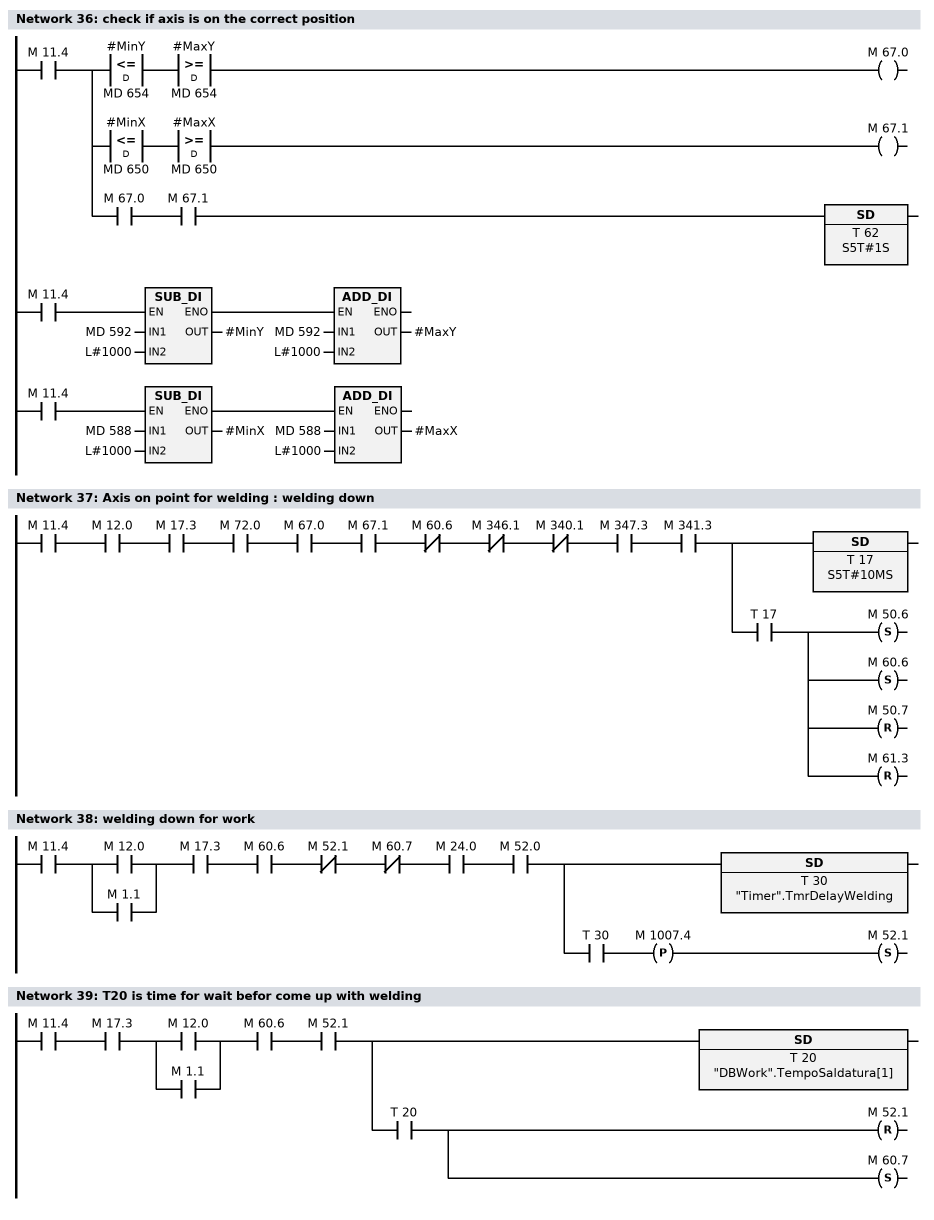
[picture p191: FC14 - AUTOMATIC networks 36-39]
NETWORK
TITLE = check if axis is on the correct position
      A     M 11.4;
      =     L 16.0;
      A(;
      A     L 16.0;
      JNB   _00e;
      L     MD 592;
      L     L#1000;
      -D;
      T     #MinY;
      AN    OV;
      SAVE;
      CLR;
_00e: A     BR;
      );
      JNB   _00f;
      L     MD 592;
      L     L#1000;
      +D;
      T     #MaxY;
_00f: NOP   0;
      A(;
      A     L 16.0;
      JNB   _010;
      L     MD 588;
      L     L#1000;
      -D;
      T     #MinX;
      AN    OV;
      SAVE;
      CLR;
_010: A     BR;
      );
      JNB   _011;
      L     MD 588;
      L     L#1000;
      +D;
      T     #MaxX;
_011: NOP   0;
      A     L 16.0;
      A(;
      L     #MinY;
      L     MD 654;
      <=D;
      );
      A(;
      L     #MaxY;
      L     MD 654;
      >=D;
      );
      =     M 67.0;
      A     L 16.0;
      A(;
      L     #MinX;
      L     MD 650;
      <=D;
      );
      A(;
      L     #MaxX;
      L     MD 650;
      >=D;
      );
      =     M 67.1;
      A     L 16.0;
      A     M 67.0;
      A     M 67.1;
      L     S5T#1S;
      SD    T 62;
NETWORK
TITLE = Axis on point for welding : welding down
//Saldatore giù
      A     M 11.4;
      A     M 12.0;
      A     M 17.3;
      A     M 72.0;
      A     M 67.0;
      A     M 67.1;
      AN    M 60.6;
      AN    M 346.1;
      AN    M 340.1;
      A     M 347.3;
      A     M 341.3;
      =     L 16.0;
      A     L 16.0;
      BLD   102;
      L     S5T#10MS;
      SD    T 17;
      A     L 16.0;
      A     T 17;
      S     M 50.6;
      S     M 60.6;
      R     M 50.7;
      R     M 61.3;
NETWORK
TITLE = welding down for work
//saldatore giu per saldatura
      A     M 11.4;
      A(;
      O     M 12.0;
      O     M 1.1;
      );
      A     M 17.3;
      A     M 60.6;
      AN    M 52.1;
      AN    M 60.7;
      A     M 24.0;
      A     M 52.0;
      =     L 16.0;
      A     L 16.0;
      BLD   102;
      L     "Timer".TmrDelayWelding;
      SD    T 30;
      A     L 16.0;
      A     T 30;
      FP    M 1007.4;
      S     M 52.1;
NETWORK
TITLE = T20 is time for wait befor come up with welding
//Resto un tempo T20 sul punto saldato prima di rialzare la torcia
      A     M 11.4;
      A     M 17.3;
      A(;
      O     M 12.0;
      O     M 1.1;
      );
      A     M 60.6;
      A     M 52.1;
      =     L 16.0;
      A     L 16.0;
      BLD   102;
      L     "DBWork".TempoSaldatura[1];
      SD    T 20;
      A     L 16.0;
      A     T 20;
      R     M 52.1;
      S     M 60.7;
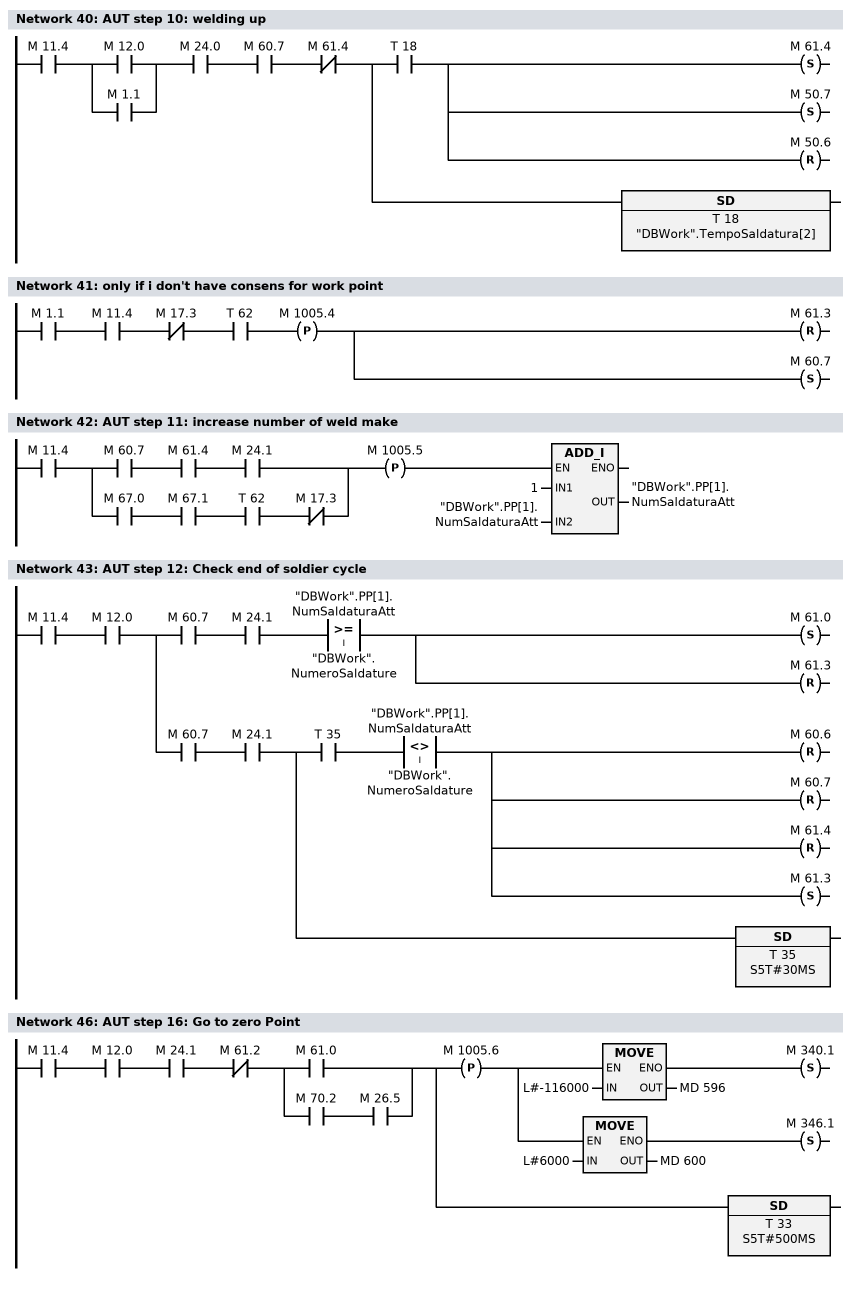
NETWORK
TITLE = AUT step 10: welding up
      A     M 11.4;
      A(;
      O     M 12.0;
      O     M 1.1;
      );
      A     M 24.0;
      A     M 60.7;
      AN    M 61.4;
      =     L 16.0;
      A     L 16.0;
      A     T 18;
      S     M 61.4;
      S     M 50.7;
      R     M 50.6;
      A     L 16.0;
      BLD   102;
      L     "DBWork".TempoSaldatura[2];
      SD    T 18;
NETWORK
TITLE = only if i don't have consens for work point
      A     M 1.1;
      A     M 11.4;
      AN    M 17.3;
      A     T 62;
      FP    M 1005.4;
      R     M 61.3;
      S     M 60.7;
NETWORK
TITLE = AUT step 11: increase number of weld make
//incremento il numero di saldature effettuate
      A     M 11.4;
      A(;
      A     M 60.7;
      A     M 61.4;
      A     M 24.1;
      O;
      A     M 67.0;
      A     M 67.1;
      A     T 62;
      AN    M 17.3;
      );
      FP    M 1005.5;
      JNB   _012;
      L     1;
      L     "DBWork".PP[1].NumSaldaturaAtt;
      +I;
      T     "DBWork".PP[1].NumSaldaturaAtt;
_012: NOP   0;
NETWORK
TITLE = AUT step 12: Check end of soldier cycle 
//aspetto per il passaggio delle coorddinate al simodrive
      A     M 11.4;
      A     M 12.0;
      =     L 16.0;
      A     L 16.0;
      A     M 60.7;
      A     M 24.1;
      A(;
      L     "DBWork".PP[1].NumSaldaturaAtt;
      L     "DBWork".NumeroSaldature;
      >=I;
      );
      S     M 61.0;
      R     M 61.3;
      A     L 16.0;
      A     M 60.7;
      A     M 24.1;
      =     L 16.1;
      A     L 16.1;
      A     T 35;
      A(;
      L     "DBWork".PP[1].NumSaldaturaAtt;
      L     "DBWork".NumeroSaldature;
      <>I;
      );
      R     M 60.6;
      R     M 60.7;
      R     M 61.4;
      S     M 61.3;
      A     L 16.1;
      BLD   102;
      L     S5T#30MS;
      SD    T 35;
NETWORK
TITLE =
NETWORK
TITLE =
NETWORK
TITLE = AUT step 16: Go to zero Point
      A     M 11.4;
      A     M 12.0;
      A     M 24.1;
      AN    M 61.2;
      A(;
      O     M 61.0;
      O;
      A     M 70.2;
      A     M 26.5;
      );
      =     L 16.0;
      A     L 16.0;
      FP    M 1005.6;
      =     L 16.1;
      A     L 16.1;
      JNB   _013;
      L     L#-116000;
      T     MD 596;
      SET;
      SAVE;
      CLR;
_013: A     BR;
      S     M 340.1;
      A     L 16.1;
      JNB   _014;
      L     L#6000;
      T     MD 600;
      SET;
      SAVE;
      CLR;
_014: A     BR;
      S     M 346.1;
      A     L 16.0;
      BLD   102;
      L     S5T#500MS;
      SD    T 33;
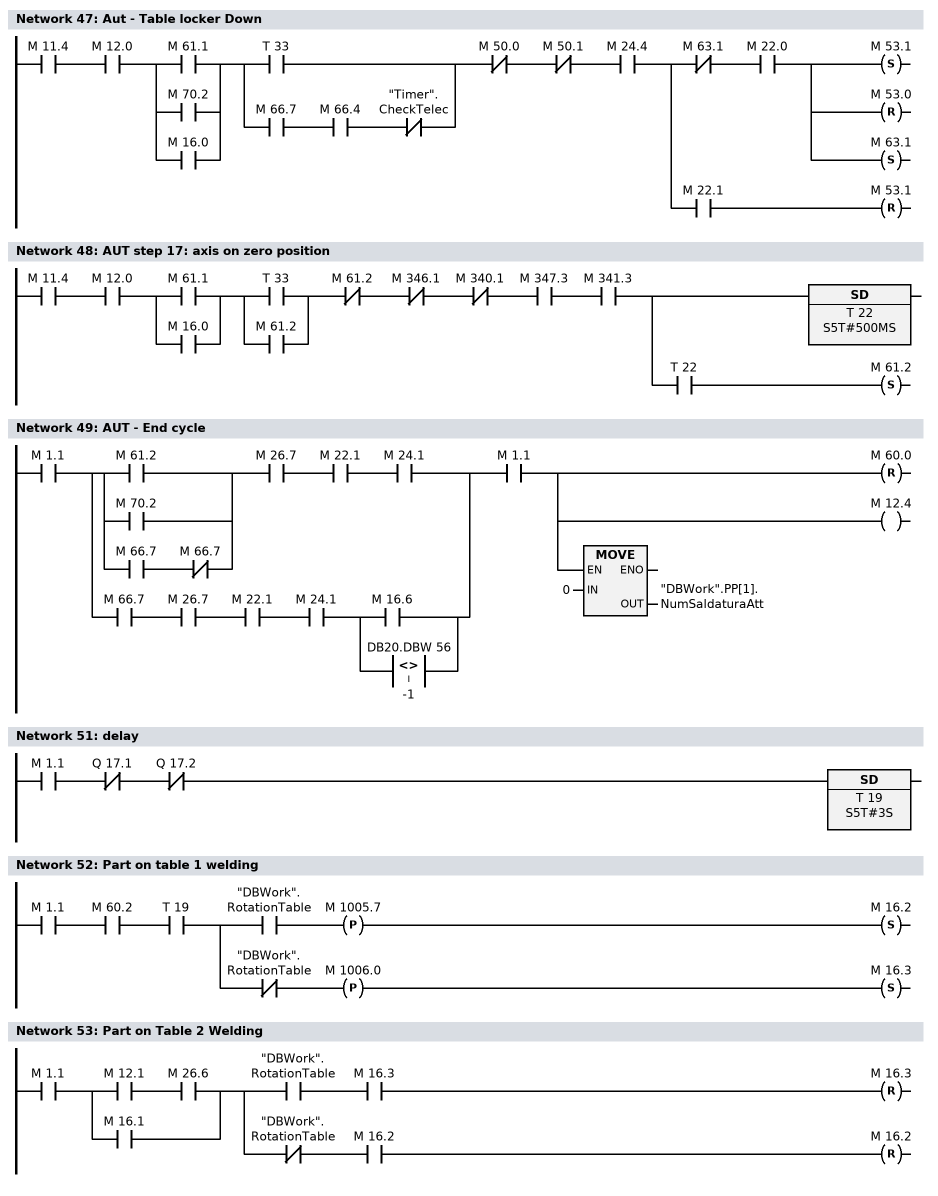
NETWORK
TITLE = Aut - Table locker Down
//Table cyclinder Low
      A     M 11.4;
      A     M 12.0;
      A(;
      O     M 61.1;
      O     M 70.2;
      O     M 16.0;
      );
      A(;
      O     T 33;
      O;
      A     M 66.7;
      A     M 66.4;
      AN    "Timer".CheckTelec;
      );
      AN    M 50.0;
      AN    M 50.1;
      A     M 24.4;
      =     L 16.0;
      A     L 16.0;
      AN    M 63.1;
      A     M 22.0;
      S     M 53.1;
      R     M 53.0;
      S     M 63.1;
      A     L 16.0;
      A     M 22.1;
      R     M 53.1;
NETWORK
TITLE = AUT step 17: axis on zero position
      A     M 11.4;
      A     M 12.0;
      A(;
      O     M 61.1;
      O     M 16.0;
      );
      A(;
      O     T 33;
      O     M 61.2;
      );
      AN    M 61.2;
      AN    M 346.1;
      AN    M 340.1;
      A     M 347.3;
      A     M 341.3;
      =     L 16.0;
      A     L 16.0;
      BLD   102;
      L     S5T#500MS;
      SD    T 22;
      A     L 16.0;
      A     T 22;
      S     M 61.2;
NETWORK
TITLE = AUT - End cycle
      A     M 1.1;
      A(;
      A(;
      O     M 61.2;
      O     M 70.2;
      O;
      A     M 66.7;
      AN    M 66.7;
      );
      A     M 26.7;
      A     M 22.1;
      A     M 24.1;
      O;
      A     M 66.7;
      A     M 26.7;
      A     M 22.1;
      A     M 24.1;
      A(;
      O     M 16.6;
      O(;
      L     DB20.DBW 56;
      L     -1;
      <>I;
      );
      );
      );
      A     M 1.1;
      =     L 16.0;
      A     L 16.0;
      BLD   102;
      R     M 60.0;
      A     L 16.0;
      BLD   102;
      =     M 12.4;
      A     L 16.0;
      JNB   _015;
      L     0;
      T     "DBWork".PP[1].NumSaldaturaAtt;
_015: NOP   0;
NETWORK
TITLE =
NETWORK
TITLE = delay
      A     M 1.1;
      AN    Q 17.1;
      AN    Q 17.2;
      L     S5T#3S;
      SD    T 19;
NETWORK
TITLE = Part on table 1 welding
      A     M 1.1;
      A     M 60.2;
      A     T 19;
      =     L 16.0;
      A     L 16.0;
      A     "DBWork".RotationTable;
      FP    M 1005.7;
      S     M 16.2;
      A     L 16.0;
      AN    "DBWork".RotationTable;
      FP    M 1006.0;
      S     M 16.3;
NETWORK
TITLE = Part on Table 2 Welding
      A     M 1.1;
      A(;
      A     M 12.1;
      A     M 26.6;
      O     M 16.1;
      );
      =     L 16.0;
      A     L 16.0;
      A     "DBWork".RotationTable;
      A     M 16.3;
      R     M 16.3;
      A     L 16.0;
      AN    "DBWork".RotationTable;
      A     M 16.2;
      R     M 16.2;
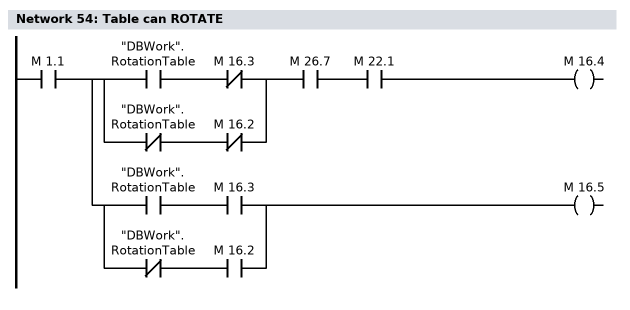
NETWORK
TITLE = Table can ROTATE
      A     M 1.1;
      =     L 16.0;
      A     L 16.0;
      A(;
      A     "DBWork".RotationTable;
      AN    M 16.3;
      O;
      AN    "DBWork".RotationTable;
      AN    M 16.2;
      );
      A     M 26.7;
      A     M 22.1;
      =     M 16.4;
      A     L 16.0;
      A(;
      A     "DBWork".RotationTable;
      A     M 16.3;
      O;
      AN    "DBWork".RotationTable;
      A     M 16.2;
      );
      =     M 16.5;
END_FUNCTION

FUNCTION "FC16 - ALARMS" : VOID	// FC 16
TITLE = Alarms management
VERSION : 0.1
VAR_TEMP
  tempBOOL : BOOL ;
END_VAR
BEGIN
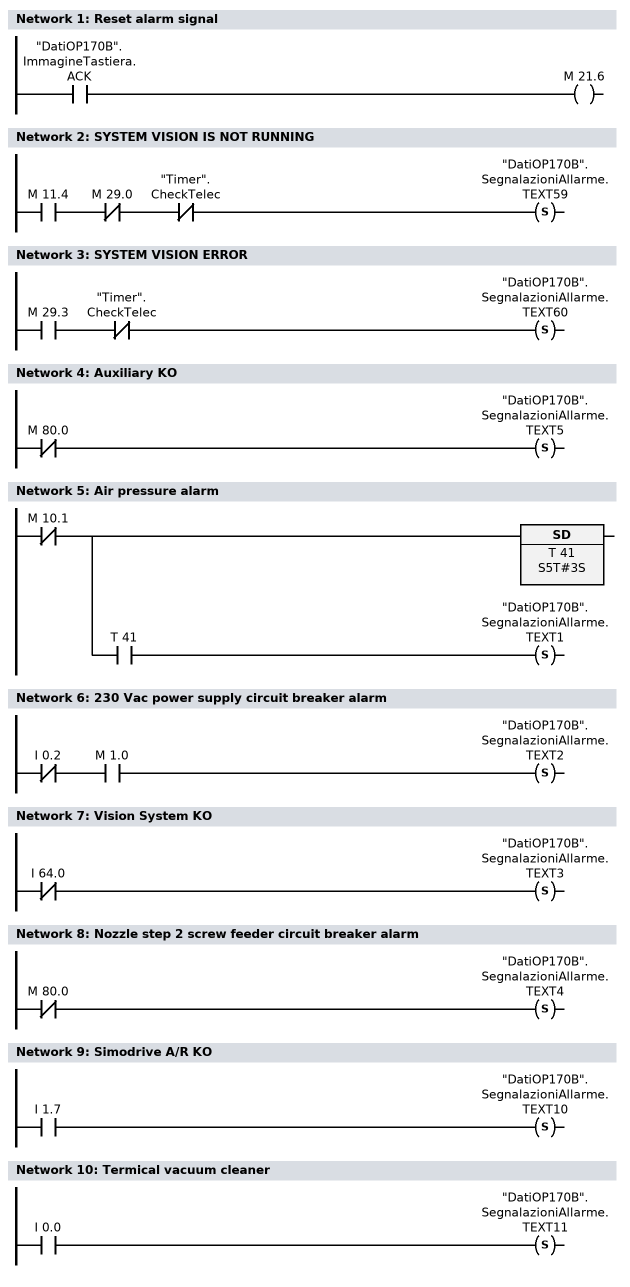
NETWORK
TITLE = Reset alarm signal
      A     "DatiOP170B".ImmagineTastiera.ACK;
      =     M 21.6;
NETWORK
TITLE = SYSTEM VISION IS NOT RUNNING
      A     M 11.4;
      AN    M 29.0;
      AN    "Timer".CheckTelec;
      S     "DatiOP170B".SegnalazioniAllarme.TEXT59;
NETWORK
TITLE = SYSTEM VISION ERROR
      A     M 29.3;
      AN    "Timer".CheckTelec;
      S     "DatiOP170B".SegnalazioniAllarme.TEXT60;
NETWORK
TITLE = Auxiliary KO
      AN    M 80.0;
      S     "DatiOP170B".SegnalazioniAllarme.TEXT5;
NETWORK
TITLE = Air pressure alarm
      AN    M 10.1;
      =     L 1.0;
      A     L 1.0;
      BLD   102;
      L     S5T#3S;
      SD    T 41;
      A     L 1.0;
      A     T 41;
      S     "DatiOP170B".SegnalazioniAllarme.TEXT1;
NETWORK
TITLE = 230 Vac power supply circuit breaker alarm
      AN    I 0.2;
      A     M 1.0;
      S     "DatiOP170B".SegnalazioniAllarme.TEXT2;
NETWORK
TITLE = Vision System KO
      AN    I 64.0;
      S     "DatiOP170B".SegnalazioniAllarme.TEXT3;
NETWORK
TITLE = Nozzle step 2 screw feeder circuit breaker alarm
      AN    M 80.0;
      S     "DatiOP170B".SegnalazioniAllarme.TEXT4;
NETWORK
TITLE = Simodrive A/R KO
      A     I 1.7;
      S     "DatiOP170B".SegnalazioniAllarme.TEXT10;
NETWORK
TITLE = Termical vacuum cleaner
      A     I 0.0;
      S     "DatiOP170B".SegnalazioniAllarme.TEXT11;
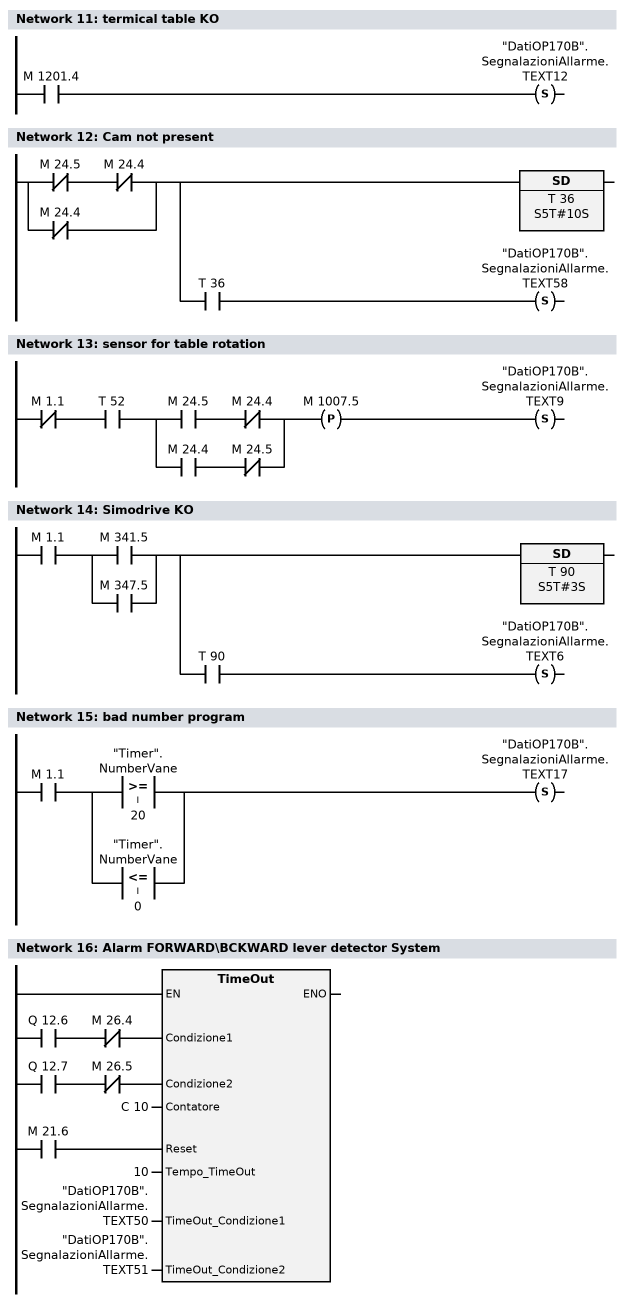
NETWORK
TITLE = termical table KO
      A     M 1201.4;
      S     "DatiOP170B".SegnalazioniAllarme.TEXT12;
NETWORK
TITLE = Cam not present
      AN    M 24.5;
      AN    M 24.4;
      ON    M 24.4;
      =     L 1.0;
      A     L 1.0;
      BLD   102;
      L     S5T#10S;
      SD    T 36;
      A     L 1.0;
      A     T 36;
      S     "DatiOP170B".SegnalazioniAllarme.TEXT58;
NETWORK
TITLE = sensor for table rotation
      AN    M 1.1;
      A     T 52;
      A(;
      A     M 24.5;
      AN    M 24.4;
      O;
      A     M 24.4;
      AN    M 24.5;
      );
      FP    M 1007.5;
      S     "DatiOP170B".SegnalazioniAllarme.TEXT9;
NETWORK
TITLE = Simodrive KO
//press ack button
      A     M 1.1;
      A(;
      O     M 341.5;
      O     M 347.5;
      );
      =     L 1.0;
      A     L 1.0;
      BLD   102;
      L     S5T#3S;
      SD    T 90;
      A     L 1.0;
      A     T 90;
      S     "DatiOP170B".SegnalazioniAllarme.TEXT6;
NETWORK
TITLE = bad number program
      A     M 1.1;
      A(;
      O(;
      L     "Timer".NumberVane;
      L     20;
      >=I;
      );
      O(;
      L     "Timer".NumberVane;
      L     0;
      <=I;
      );
      );
      S     "DatiOP170B".SegnalazioniAllarme.TEXT17;
NETWORK
TITLE = Alarm FORWARD\BCKWARD lever detector System
      A     Q 12.6;
      AN    M 26.4;
      =     L 1.0;
      BLD   103;
      A     Q 12.7;
      AN    M 26.5;
      =     L 1.1;
      BLD   103;
      A     M 21.6;
      =     L 1.2;
      BLD   103;
      CALL  "TimeOut" (
           Condizione1              := L 1.0,
           Condizione2              := L 1.1,
           Contatore                := C 10,
           Reset                    := L 1.2,
           Tempo_TimeOut            := 10,
           TimeOut_Condizione1      := "DatiOP170B".SegnalazioniAllarme.TEXT50,
           TimeOut_Condizione2      := "DatiOP170B".SegnalazioniAllarme.TEXT51);
      NOP   0;
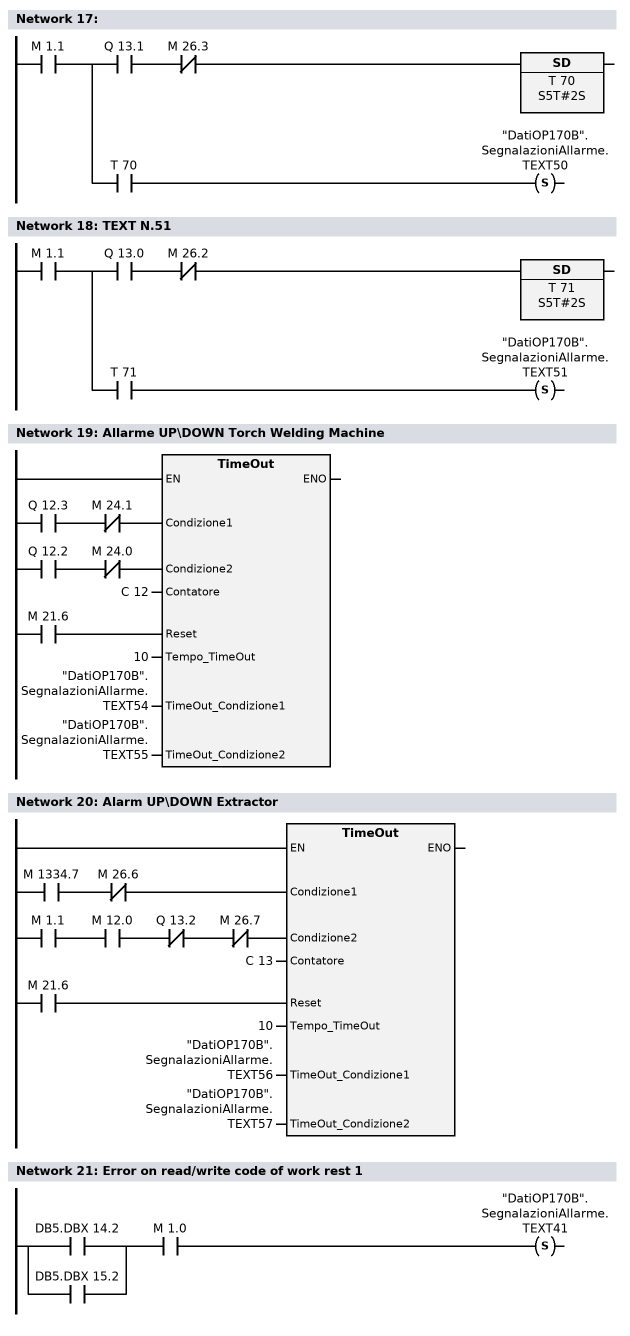
NETWORK
TITLE =
      A     M 1.1;
      =     L 1.0;
      A     L 1.0;
      A     Q 13.1;
      AN    M 26.3;
      L     S5T#2S;
      SD    T 70;
      A     L 1.0;
      A     T 70;
      S     "DatiOP170B".SegnalazioniAllarme.TEXT50;
NETWORK
TITLE = TEXT N.51
      A     M 1.1;
      =     L 1.0;
      A     L 1.0;
      A     Q 13.0;
      AN    M 26.2;
      L     S5T#2S;
      SD    T 71;
      A     L 1.0;
      A     T 71;
      S     "DatiOP170B".SegnalazioniAllarme.TEXT51;
NETWORK
TITLE = Allarme UP\DOWN Torch Welding Machine
      A     Q 12.3;
      AN    M 24.1;
      =     L 1.0;
      BLD   103;
      A     Q 12.2;
      AN    M 24.0;
      =     L 1.1;
      BLD   103;
      A     M 21.6;
      =     L 1.2;
      BLD   103;
      CALL  "TimeOut" (
           Condizione1              := L 1.0,
           Condizione2              := L 1.1,
           Contatore                := C 12,
           Reset                    := L 1.2,
           Tempo_TimeOut            := 10,
           TimeOut_Condizione1      := "DatiOP170B".SegnalazioniAllarme.TEXT54,
           TimeOut_Condizione2      := "DatiOP170B".SegnalazioniAllarme.TEXT55);
      NOP   0;
NETWORK
TITLE = Alarm UP\DOWN Extractor
      A     M 1334.7;
      AN    M 26.6;
      =     L 1.0;
      BLD   103;
      A     M 1.1;
      A     M 12.0;
      AN    Q 13.2;
      AN    M 26.7;
      =     L 1.1;
      BLD   103;
      A     M 21.6;
      =     L 1.2;
      BLD   103;
      CALL  "TimeOut" (
           Condizione1              := L 1.0,
           Condizione2              := L 1.1,
           Contatore                := C 13,
           Reset                    := L 1.2,
           Tempo_TimeOut            := 10,
           TimeOut_Condizione1      := "DatiOP170B".SegnalazioniAllarme.TEXT56,
           TimeOut_Condizione2      := "DatiOP170B".SegnalazioniAllarme.TEXT57);
      NOP   0;
NETWORK
TITLE = Error on read/write code of work rest 1
      A(;
      O     DB5.DBX 14.2;
      O     DB5.DBX 15.2;
      );
      A     M 1.0;
      S     "DatiOP170B".SegnalazioniAllarme.TEXT41;
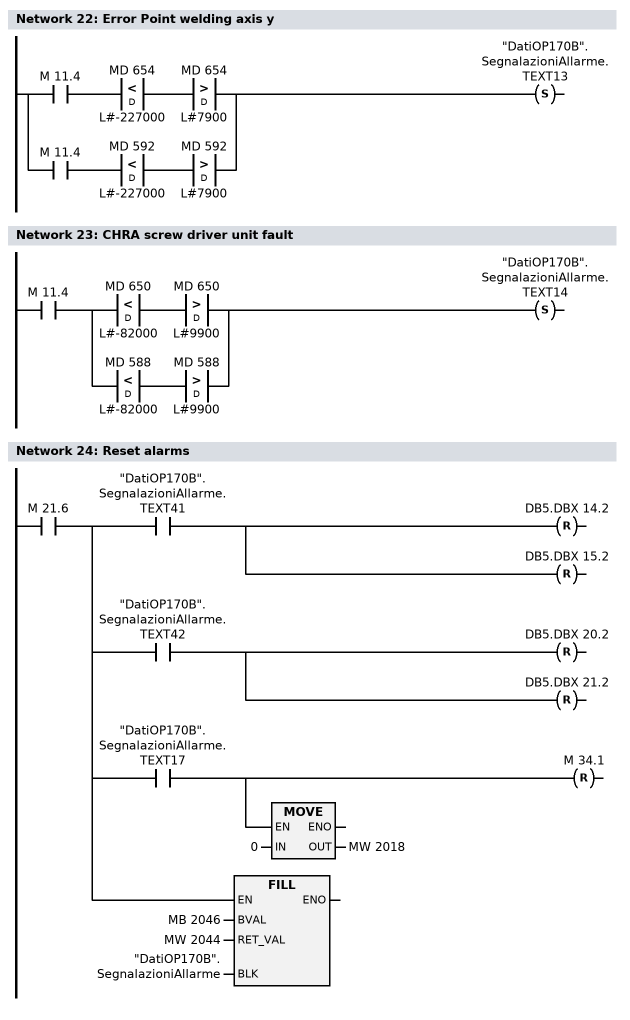
NETWORK
TITLE = Error Point welding axis y
      A     M 11.4;
      A(;
      L     MD 654;
      L     L#-227000;
      <D;
      );
      A(;
      L     MD 654;
      L     L#7900;
      >D;
      );
      O;
      A     M 11.4;
      A(;
      L     MD 592;
      L     L#-227000;
      <D;
      );
      A(;
      L     MD 592;
      L     L#7900;
      >D;
      );
      S     "DatiOP170B".SegnalazioniAllarme.TEXT13;
NETWORK
TITLE = CHRA screw driver unit fault
      A     M 11.4;
      A(;
      A(;
      L     MD 650;
      L     L#-82000;
      <D;
      );
      A(;
      L     MD 650;
      L     L#9900;
      >D;
      );
      O;
      A(;
      L     MD 588;
      L     L#-82000;
      <D;
      );
      A(;
      L     MD 588;
      L     L#9900;
      >D;
      );
      );
      S     "DatiOP170B".SegnalazioniAllarme.TEXT14;
NETWORK
TITLE = Reset alarms
      A     M 21.6;
      =     L 1.0;
      A     L 1.0;
      A     "DatiOP170B".SegnalazioniAllarme.TEXT41;
      R     DB5.DBX 14.2;
      R     DB5.DBX 15.2;
      A     L 1.0;
      A     "DatiOP170B".SegnalazioniAllarme.TEXT42;
      R     DB5.DBX 20.2;
      R     DB5.DBX 21.2;
      A     L 1.0;
      A     "DatiOP170B".SegnalazioniAllarme.TEXT17;
      =     L 1.1;
      A     L 1.1;
      BLD   102;
      R     M 34.1;
      A     L 1.1;
      JNB   _001;
      L     0;
      T     MW 2018;
_001: NOP   0;
      A     L 1.0;
      JNB   _002;
      CALL  "FILL" (
           BVAL                     := MB 2046,
           RET_VAL                  := MW 2044,
           BLK                      := "DatiOP170B".SegnalazioniAllarme);
_002: NOP   0;
NETWORK
TITLE = Spacer circular feeder empty
      CLR;
      =     "DatiOP170B".SegnalazioniAllarme.TEXT15;
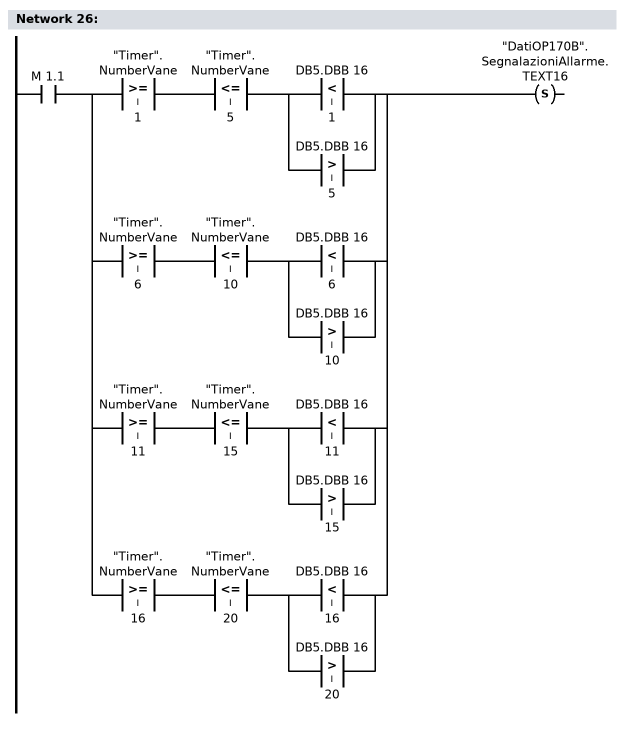
NETWORK
TITLE =
      A     M 1.1;
      A(;
      A(;
      L     "Timer".NumberVane;
      L     1;
      >=I;
      );
      A(;
      L     "Timer".NumberVane;
      L     5;
      <=I;
      );
      A(;
      O(;
      L     DB5.DBB 16;
      L     1;
      <I;
      );
      O(;
      L     DB5.DBB 16;
      L     5;
      >I;
      );
      );
      O;
      A(;
      L     "Timer".NumberVane;
      L     6;
      >=I;
      );
      A(;
      L     "Timer".NumberVane;
      L     10;
      <=I;
      );
      A(;
      O(;
      L     DB5.DBB 16;
      L     6;
      <I;
      );
      O(;
      L     DB5.DBB 16;
      L     10;
      >I;
      );
      );
      O;
      A(;
      L     "Timer".NumberVane;
      L     11;
      >=I;
      );
      A(;
      L     "Timer".NumberVane;
      L     15;
      <=I;
      );
      A(;
      O(;
      L     DB5.DBB 16;
      L     11;
      <I;
      );
      O(;
      L     DB5.DBB 16;
      L     15;
      >I;
      );
      );
      O;
      A(;
      L     "Timer".NumberVane;
      L     16;
      >=I;
      );
      A(;
      L     "Timer".NumberVane;
      L     20;
      <=I;
      );
      A(;
      O(;
      L     DB5.DBB 16;
      L     16;
      <I;
      );
      O(;
      L     DB5.DBB 16;
      L     20;
      >I;
      );
      );
      );
      S     "DatiOP170B".SegnalazioniAllarme.TEXT16;
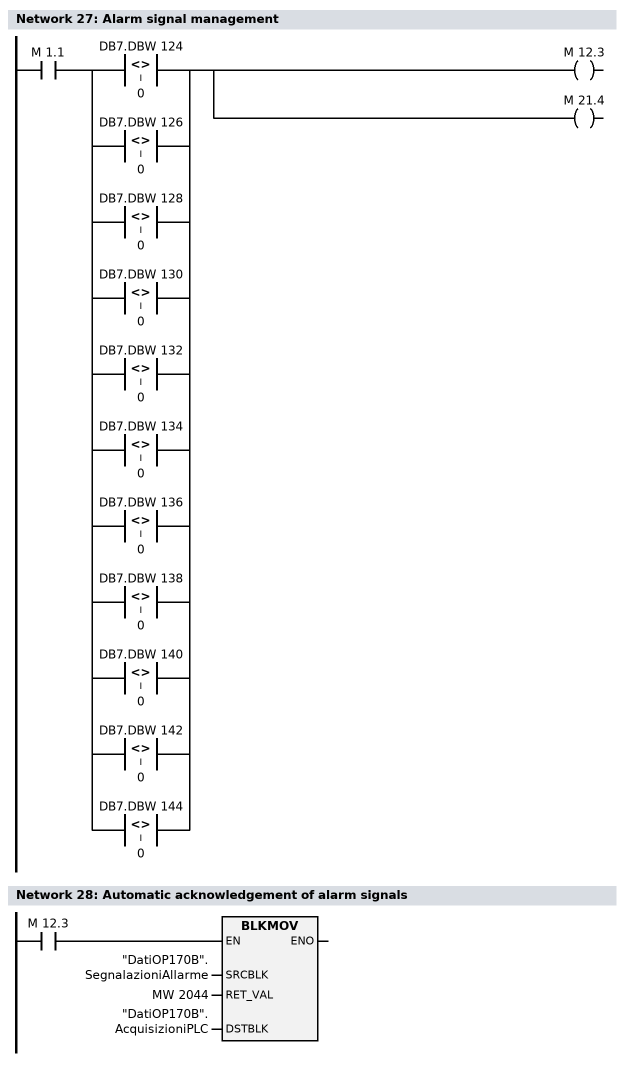
NETWORK
TITLE = Alarm signal management
      A     M 1.1;
      A(;
      O(;
      L     DB7.DBW 124;
      L     0;
      <>I;
      );
      O(;
      L     DB7.DBW 126;
      L     0;
      <>I;
      );
      O(;
      L     DB7.DBW 128;
      L     0;
      <>I;
      );
      O(;
      L     DB7.DBW 130;
      L     0;
      <>I;
      );
      O(;
      L     DB7.DBW 132;
      L     0;
      <>I;
      );
      O(;
      L     DB7.DBW 134;
      L     0;
      <>I;
      );
      O(;
      L     DB7.DBW 136;
      L     0;
      <>I;
      );
      O(;
      L     DB7.DBW 138;
      L     0;
      <>I;
      );
      O(;
      L     DB7.DBW 140;
      L     0;
      <>I;
      );
      O(;
      L     DB7.DBW 142;
      L     0;
      <>I;
      );
      O(;
      L     DB7.DBW 144;
      L     0;
      <>I;
      );
      );
      =     M 12.3;
      =     M 21.4;
NETWORK
TITLE = Automatic acknowledgement of alarm signals
      A     M 12.3;
      JNB   _003;
      CALL  "BLKMOV" (
           SRCBLK                   := "DatiOP170B".SegnalazioniAllarme,
           RET_VAL                  := MW 2044,
           DSTBLK                   := "DatiOP170B".AcquisizioniPLC);
_003: NOP   0;
END_FUNCTION

FUNCTION "FC17 - OPERATOR PANNEL" : VOID	// FC 17
TITLE = OP170B Operator Pannel Interface
VERSION : 0.1
BEGIN
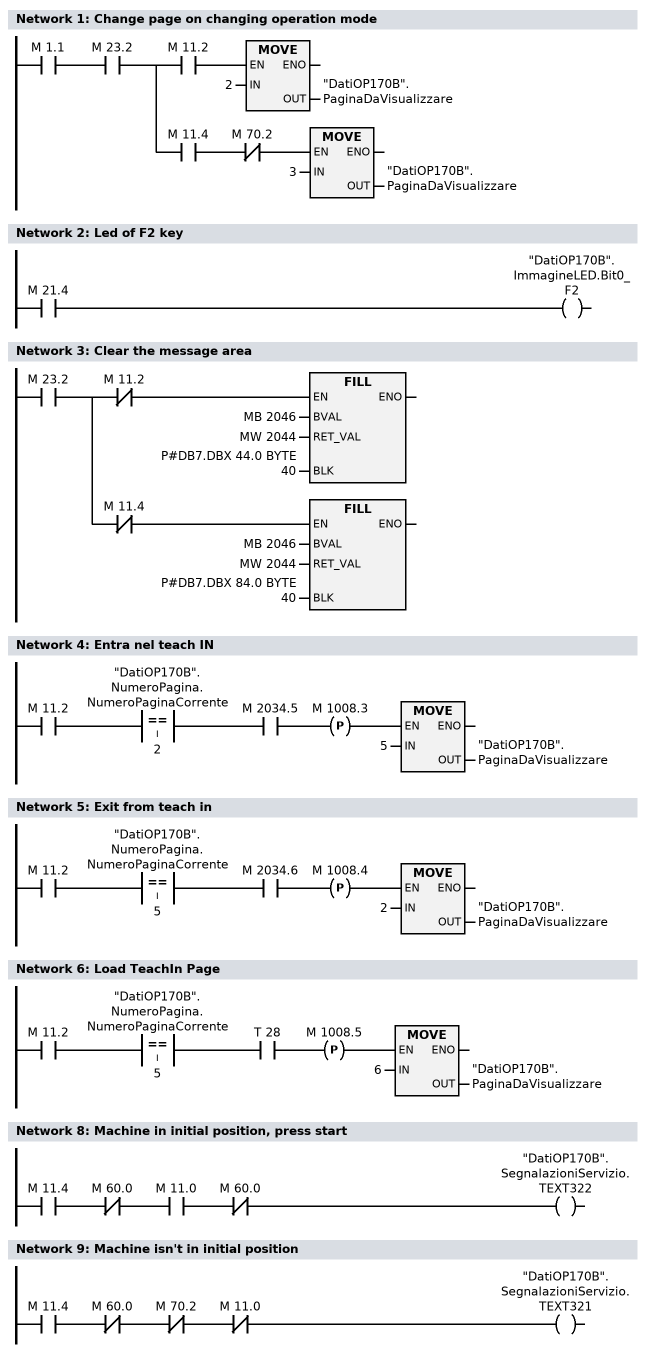
NETWORK
TITLE = Change page on changing operation mode
      A     M 1.1;
      A     M 23.2;
      =     L 0.0;
      A     L 0.0;
      A     M 11.2;
      JNB   _001;
      L     2;
      T     "DatiOP170B".PaginaDaVisualizzare;
_001: NOP   0;
      A     L 0.0;
      A     M 11.4;
      AN    M 70.2;
      JNB   _002;
      L     3;
      T     "DatiOP170B".PaginaDaVisualizzare;
_002: NOP   0;
NETWORK
TITLE = Led of F2 key
      A     M 21.4;
      =     "DatiOP170B".ImmagineLED.Bit0_F2;
NETWORK
TITLE = Clear the message area
      A     M 23.2;
      =     L 0.0;
      A     L 0.0;
      AN    M 11.2;
      JNB   _003;
      CALL  "FILL" (
           BVAL                     := MB 2046,
           RET_VAL                  := MW 2044,
           BLK                      := P#DB7.DBX 44.0 BYTE 40);
_003: NOP   0;
      A     L 0.0;
      AN    M 11.4;
      JNB   _004;
      CALL  "FILL" (
           BVAL                     := MB 2046,
           RET_VAL                  := MW 2044,
           BLK                      := P#DB7.DBX 84.0 BYTE 40);
_004: NOP   0;
NETWORK
TITLE = Entra nel teach IN
      A     M 11.2;
      A(;
      L     "DatiOP170B".NumeroPagina.NumeroPaginaCorrente;
      L     2;
      ==I;
      );
      A     M 2034.5;
      FP    M 1008.3;
      JNB   _005;
      L     5;
      T     "DatiOP170B".PaginaDaVisualizzare;
_005: NOP   0;
NETWORK
TITLE = Exit from teach in
      A     M 11.2;
      A(;
      L     "DatiOP170B".NumeroPagina.NumeroPaginaCorrente;
      L     5;
      ==I;
      );
      A     M 2034.6;
      FP    M 1008.4;
      JNB   _006;
      L     2;
      T     "DatiOP170B".PaginaDaVisualizzare;
_006: NOP   0;
NETWORK
TITLE = Load TeachIn Page
//Aspetto il T28 in modo tale da lanciare il comando agli assi
      A     M 11.2;
      A(;
      L     "DatiOP170B".NumeroPagina.NumeroPaginaCorrente;
      L     5;
      ==I;
      );
      A     T 28;
      FP    M 1008.5;
      JNB   _007;
      L     6;
      T     "DatiOP170B".PaginaDaVisualizzare;
_007: NOP   0;
NETWORK
TITLE =
NETWORK
TITLE = Machine in initial position, press start
      A     M 11.4;
      AN    M 60.0;
      A     M 11.0;
      AN    M 60.0;
      =     "DatiOP170B".SegnalazioniServizio.TEXT322;
NETWORK
TITLE = Machine isn't in initial position
      A     M 11.4;
      AN    M 60.0;
      AN    M 70.2;
      AN    M 11.0;
      =     "DatiOP170B".SegnalazioniServizio.TEXT321;
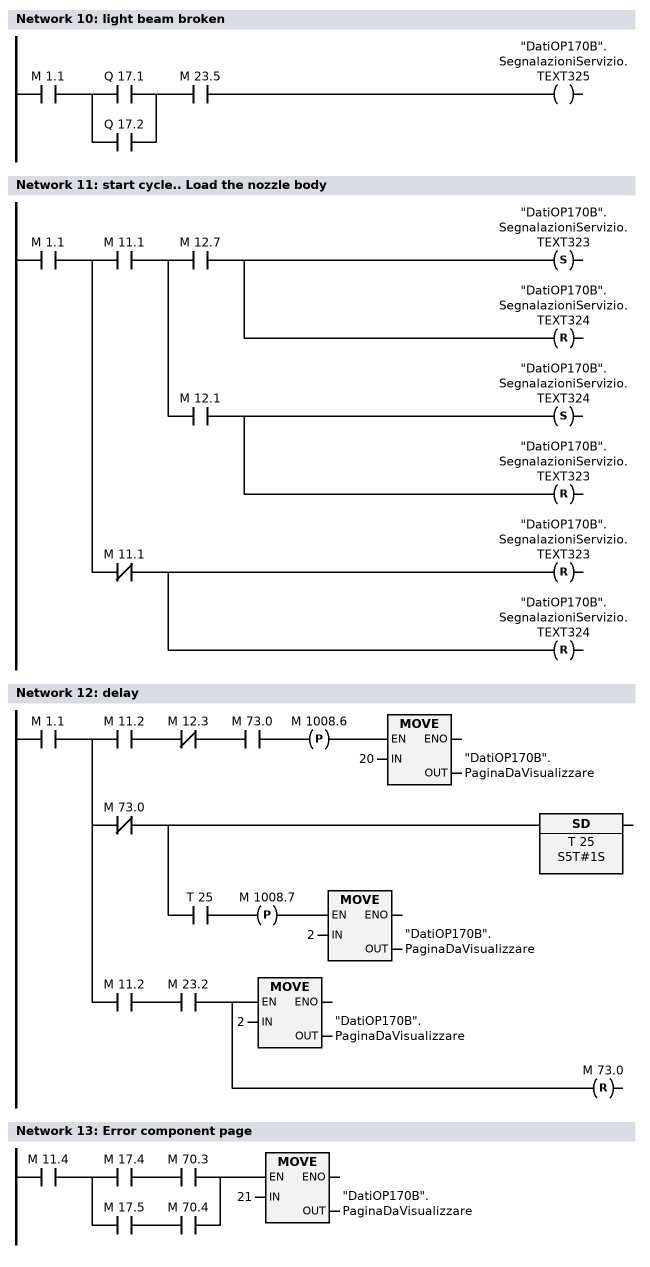
NETWORK
TITLE = light beam broken
      A     M 1.1;
      A(;
      O     Q 17.1;
      O     Q 17.2;
      );
      A     M 23.5;
      =     "DatiOP170B".SegnalazioniServizio.TEXT325;
NETWORK
TITLE = start cycle.. Load the nozzle body
      A     M 1.1;
      =     L 0.0;
      A     L 0.0;
      A     M 11.1;
      =     L 0.1;
      A     L 0.1;
      A     M 12.7;
      S     "DatiOP170B".SegnalazioniServizio.TEXT323;
      R     "DatiOP170B".SegnalazioniServizio.TEXT324;
      A     L 0.1;
      A     M 12.1;
      S     "DatiOP170B".SegnalazioniServizio.TEXT324;
      R     "DatiOP170B".SegnalazioniServizio.TEXT323;
      A     L 0.0;
      AN    M 11.1;
      R     "DatiOP170B".SegnalazioniServizio.TEXT323;
      R     "DatiOP170B".SegnalazioniServizio.TEXT324;
NETWORK
TITLE = delay
//Page of repositioning
      A     M 1.1;
      =     L 0.0;
      A     L 0.0;
      A     M 11.2;
      AN    M 12.3;
      A     M 73.0;
      FP    M 1008.6;
      JNB   _008;
      L     20;
      T     "DatiOP170B".PaginaDaVisualizzare;
_008: NOP   0;
      A     L 0.0;
      AN    M 73.0;
      =     L 0.1;
      A     L 0.1;
      BLD   102;
      L     S5T#1S;
      SD    T 25;
      A     L 0.1;
      A     T 25;
      FP    M 1008.7;
      JNB   _009;
      L     2;
      T     "DatiOP170B".PaginaDaVisualizzare;
_009: NOP   0;
      A     L 0.0;
      A     M 11.2;
      A     M 23.2;
      =     L 0.1;
      A     L 0.1;
      JNB   _00a;
      L     2;
      T     "DatiOP170B".PaginaDaVisualizzare;
_00a: NOP   0;
      A     L 0.1;
      BLD   102;
      R     M 73.0;
NETWORK
TITLE = Error component page
      A     M 11.4;
      A(;
      A     M 17.4;
      A     M 70.3;
      O;
      A     M 17.5;
      A     M 70.4;
      );
      JNB   _00b;
      L     21;
      T     "DatiOP170B".PaginaDaVisualizzare;
_00b: NOP   0;
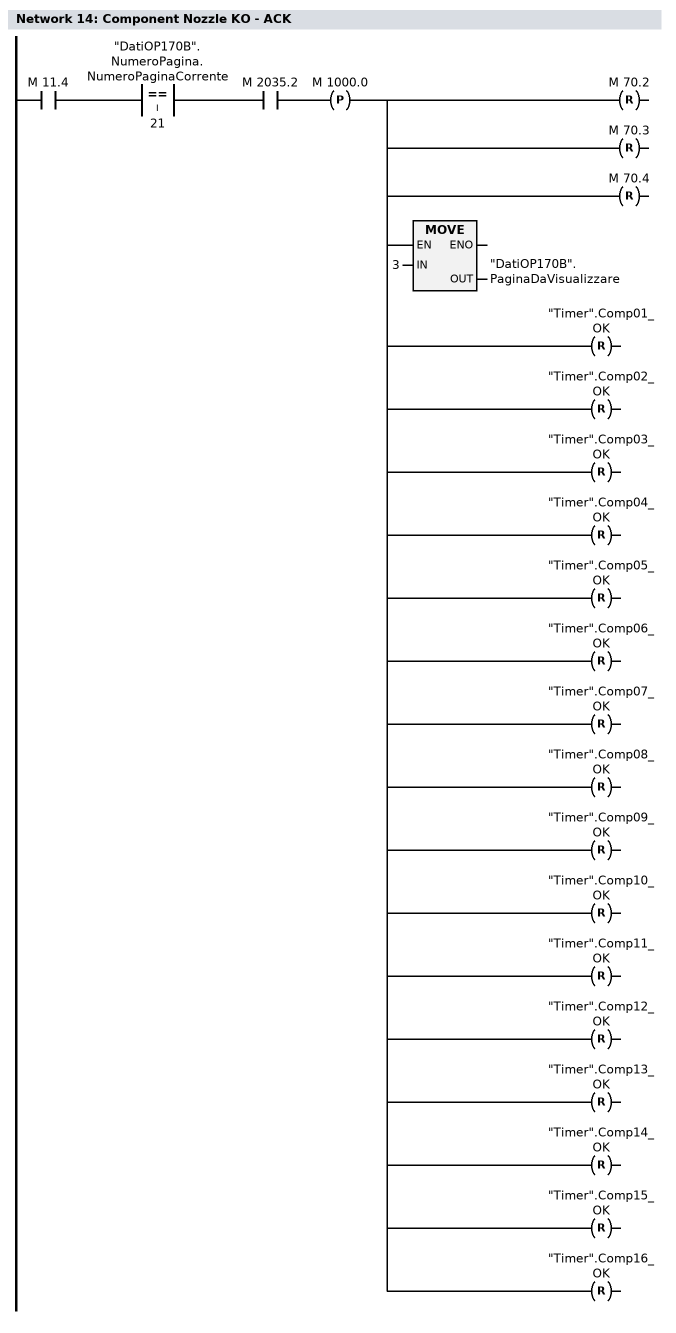
NETWORK
TITLE = Component Nozzle KO - ACK
      A     M 11.4;
      A(;
      L     "DatiOP170B".NumeroPagina.NumeroPaginaCorrente;
      L     21;
      ==I;
      );
      A     M 2035.2;
      FP    M 1000.0;
      =     L 0.0;
      A     L 0.0;
      BLD   102;
      R     M 70.2;
      A     L 0.0;
      BLD   102;
      R     M 70.3;
      A     L 0.0;
      BLD   102;
      R     M 70.4;
      A     L 0.0;
      JNB   _00c;
      L     3;
      T     "DatiOP170B".PaginaDaVisualizzare;
_00c: NOP   0;
      A     L 0.0;
      BLD   102;
      R     "Timer".Comp01_OK;
      A     L 0.0;
      BLD   102;
      R     "Timer".Comp02_OK;
      A     L 0.0;
      BLD   102;
      R     "Timer".Comp03_OK;
      A     L 0.0;
      BLD   102;
      R     "Timer".Comp04_OK;
      A     L 0.0;
      BLD   102;
      R     "Timer".Comp05_OK;
      A     L 0.0;
      BLD   102;
      R     "Timer".Comp06_OK;
      A     L 0.0;
      BLD   102;
      R     "Timer".Comp07_OK;
      A     L 0.0;
      BLD   102;
      R     "Timer".Comp08_OK;
      A     L 0.0;
      BLD   102;
      R     "Timer".Comp09_OK;
      A     L 0.0;
      BLD   102;
      R     "Timer".Comp10_OK;
      A     L 0.0;
      BLD   102;
      R     "Timer".Comp11_OK;
      A     L 0.0;
      BLD   102;
      R     "Timer".Comp12_OK;
      A     L 0.0;
      BLD   102;
      R     "Timer".Comp13_OK;
      A     L 0.0;
      BLD   102;
      R     "Timer".Comp14_OK;
      A     L 0.0;
      BLD   102;
      R     "Timer".Comp15_OK;
      A     L 0.0;
      BLD   102;
      R     "Timer".Comp16_OK;
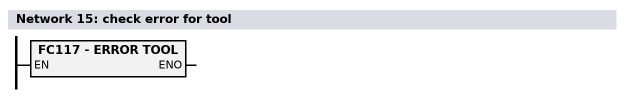
NETWORK
TITLE = check error for tool
      CALL  "FC117 - ERROR TOOL";
      NOP   0;
END_FUNCTION

FUNCTION "FC18 - OUTPUTS" : VOID	// FC 18
TITLE = Outputs management
VERSION : 0.1
BEGIN
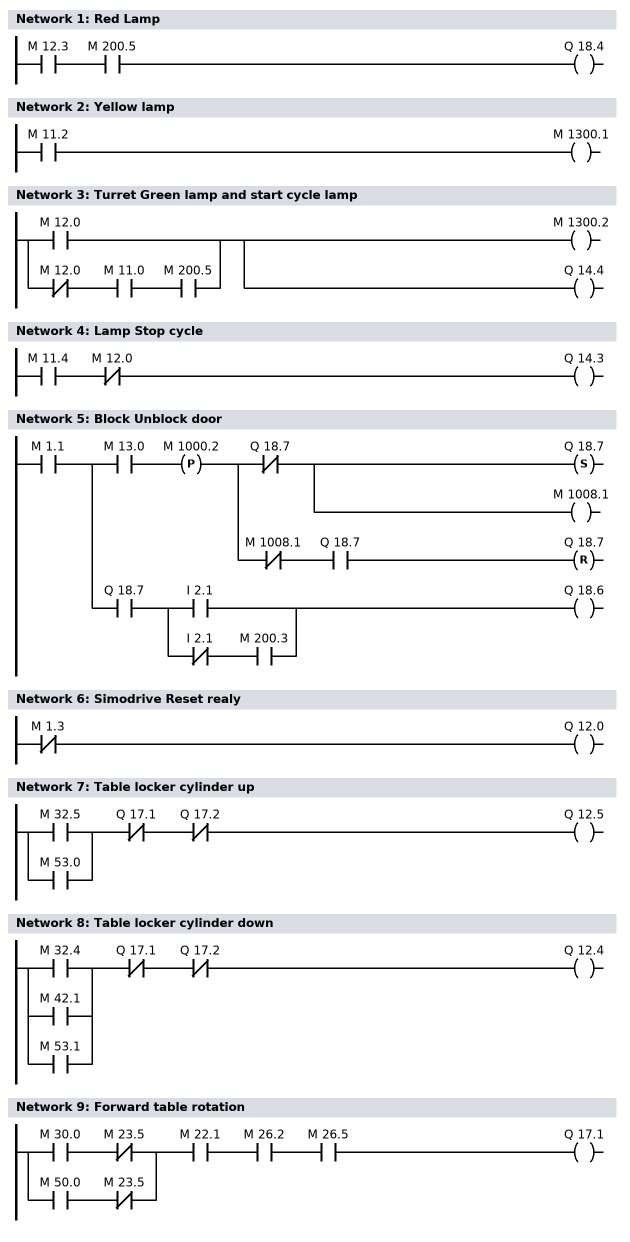
NETWORK
TITLE = Red Lamp
      A     M 12.3;
      A     M 200.5;
      =     Q 18.4;
NETWORK
TITLE = Yellow lamp
      A     M 11.2;
      =     M 1300.1;
NETWORK
TITLE = Turret Green lamp and start cycle lamp
      O     M 12.0;
      O;
      AN    M 12.0;
      A     M 11.0;
      A     M 200.5;
      =     M 1300.2;
      =     Q 14.4;
NETWORK
TITLE = Lamp Stop cycle
      A     M 11.4;
      AN    M 12.0;
      =     Q 14.3;
NETWORK
TITLE = Block Unblock door
//light ON = door lock
      A     M 1.1;
      =     L 0.0;
      A     L 0.0;
      A     M 13.0;
      FP    M 1000.2;
      =     L 0.1;
      A     L 0.1;
      AN    Q 18.7;
      S     Q 18.7;
      =     M 1008.1;
      A     L 0.1;
      AN    M 1008.1;
      A     Q 18.7;
      R     Q 18.7;
      A     L 0.0;
      A     Q 18.7;
      A(;
      O     I 2.1;
      O;
      AN    I 2.1;
      A     M 200.3;
      );
      =     Q 18.6;
NETWORK
TITLE = Simodrive Reset realy
      AN    M 1.3;
      =     Q 12.0;
NETWORK
TITLE = Table locker cylinder up
      A(;
      O     M 32.5;
      O     M 53.0;
      );
      AN    Q 17.1;
      AN    Q 17.2;
      =     Q 12.5;
NETWORK
TITLE = Table locker cylinder down
      A(;
      O     M 32.4;
      O     M 42.1;
      O     M 53.1;
      );
      AN    Q 17.1;
      AN    Q 17.2;
      =     Q 12.4;
NETWORK
TITLE = Forward table rotation
      A(;
      A     M 30.0;
      AN    M 23.5;
      O;
      A     M 50.0;
      AN    M 23.5;
      );
      A     M 22.1;
      A     M 26.2;
      A     M 26.5;
      =     Q 17.1;
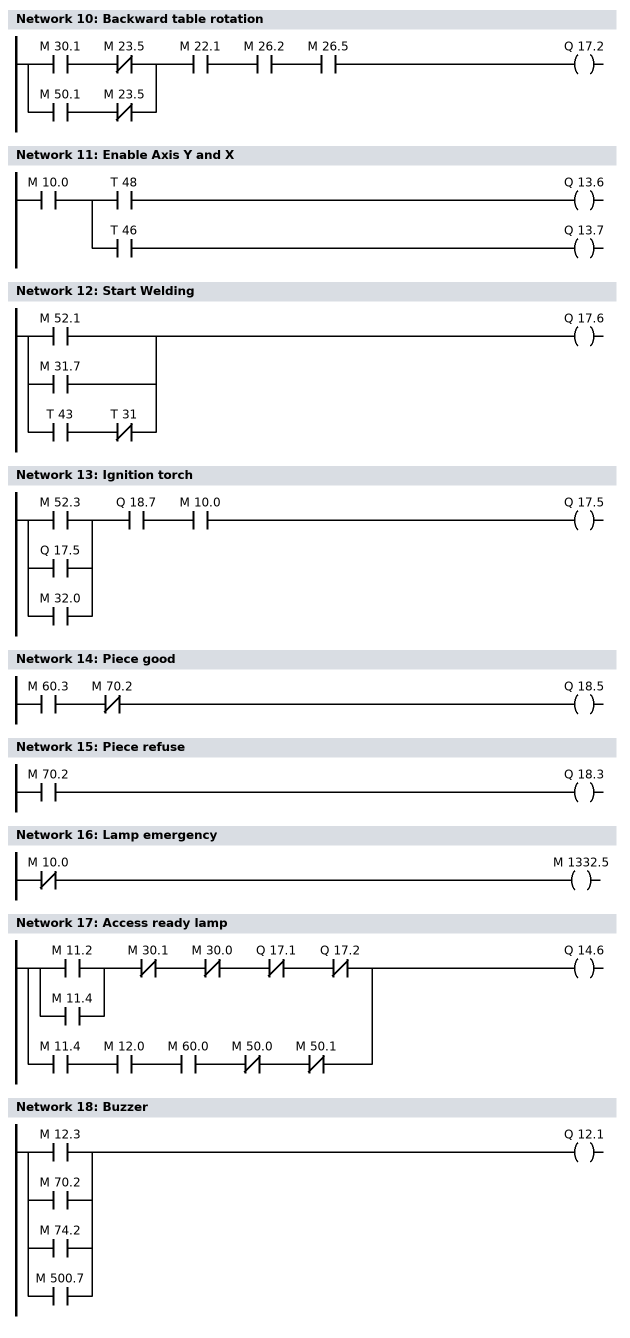
NETWORK
TITLE = Backward table rotation
      A(;
      A     M 30.1;
      AN    M 23.5;
      O;
      A     M 50.1;
      AN    M 23.5;
      );
      A     M 22.1;
      A     M 26.2;
      A     M 26.5;
      =     Q 17.2;
NETWORK
TITLE = Enable Axis Y and X
      A     M 10.0;
      =     L 0.0;
      A     L 0.0;
      A     T 48;
      =     Q 13.6;
      A     L 0.0;
      A     T 46;
      =     Q 13.7;
NETWORK
TITLE = Start Welding
      O     M 52.1;
      O     M 31.7;
      O;
      A     T 43;
      AN    T 31;
      =     Q 17.6;
NETWORK
TITLE = Ignition torch
      A(;
      O     M 52.3;
      O     Q 17.5;
      O     M 32.0;
      );
      A     Q 18.7;
      A     M 10.0;
      =     Q 17.5;
NETWORK
TITLE = Piece good
      A     M 60.3;
      AN    M 70.2;
      =     Q 18.5;
NETWORK
TITLE = Piece refuse
      A     M 70.2;
      =     Q 18.3;
NETWORK
TITLE = Lamp emergency
      AN    M 10.0;
      =     M 1332.5;
NETWORK
TITLE = Access ready lamp
      A(;
      O     M 11.2;
      O     M 11.4;
      );
      AN    M 30.1;
      AN    M 30.0;
      AN    Q 17.1;
      AN    Q 17.2;
      O;
      A     M 11.4;
      A     M 12.0;
      A     M 60.0;
      AN    M 50.0;
      AN    M 50.1;
      =     Q 14.6;
NETWORK
TITLE = Buzzer
//"Off"
      O     M 12.3;
      O     M 70.2;
      O     M 74.2;
      O     M 500.7;
      =     Q 12.1;
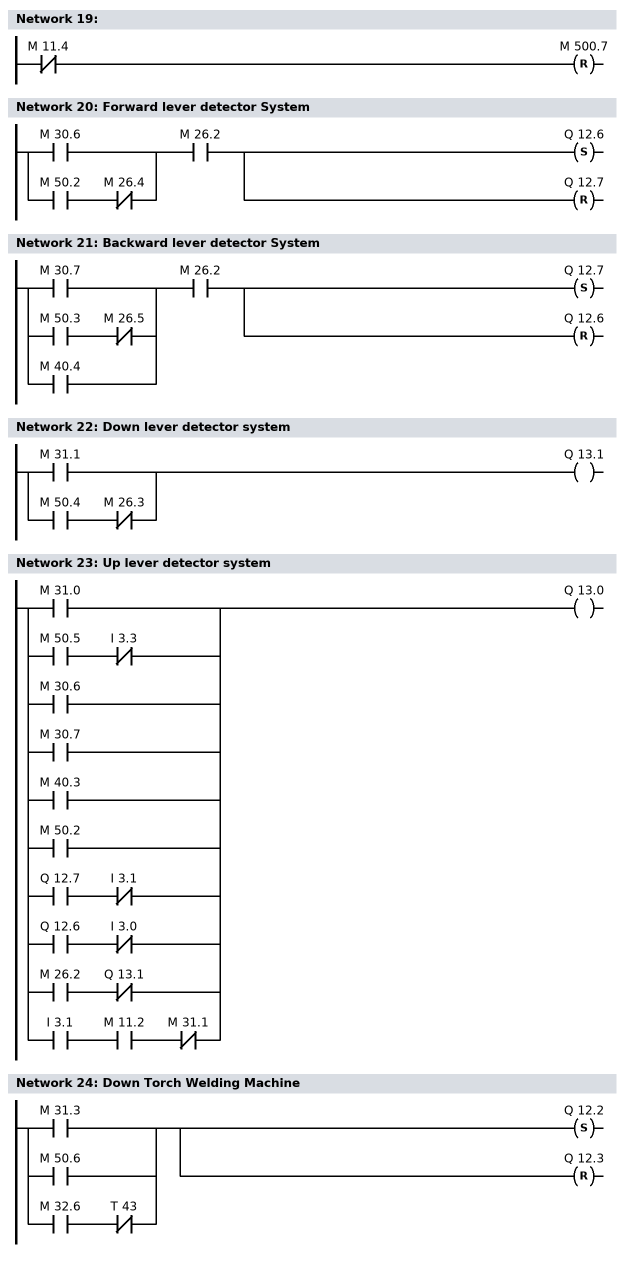
NETWORK
TITLE =
      AN    M 11.4;
      R     M 500.7;
NETWORK
TITLE = Forward lever detector System
      A(;
      O     M 30.6;
      O;
      A     M 50.2;
      AN    M 26.4;
      );
      A     M 26.2;
      S     Q 12.6;
      R     Q 12.7;
NETWORK
TITLE = Backward lever detector System
      A(;
      O     M 30.7;
      O;
      A     M 50.3;
      AN    M 26.5;
      O     M 40.4;
      );
      A     M 26.2;
      S     Q 12.7;
      R     Q 12.6;
NETWORK
TITLE = Down lever detector system
      O     M 31.1;
      O;
      A     M 50.4;
      AN    M 26.3;
      =     Q 13.1;
NETWORK
TITLE = Up lever detector system
      O     M 31.0;
      O;
      A     M 50.5;
      AN    I 3.3;
      O     M 30.6;
      O     M 30.7;
      O     M 40.3;
      O     M 50.2;
      O;
      A     Q 12.7;
      AN    I 3.1;
      O;
      A     Q 12.6;
      AN    I 3.0;
      O;
      A     M 26.2;
      AN    Q 13.1;
      O;
      A     I 3.1;
      A     M 11.2;
      AN    M 31.1;
      =     Q 13.0;
NETWORK
TITLE = Down Torch Welding Machine
      O     M 31.3;
      O     M 50.6;
      O;
      A     M 32.6;
      AN    T 43;
      S     Q 12.2;
      R     Q 12.3;
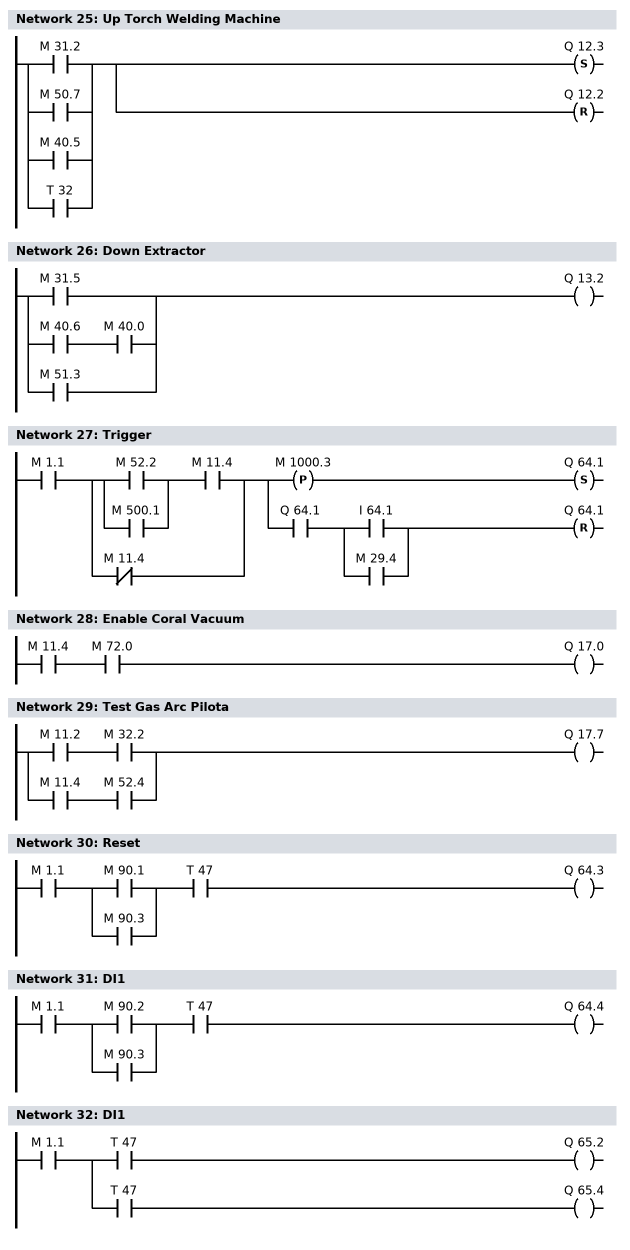
NETWORK
TITLE = Up Torch Welding Machine
      O     M 31.2;
      O     M 50.7;
      O     M 40.5;
      O     T 32;
      S     Q 12.3;
      R     Q 12.2;
NETWORK
TITLE = Down Extractor
      O     M 31.5;
      O;
      A     M 40.6;
      A     M 40.0;
      O     M 51.3;
      =     Q 13.2;
NETWORK
TITLE = Trigger
      A     M 1.1;
      A(;
      A(;
      O     M 52.2;
      O     M 500.1;
      );
      A     M 11.4;
      ON    M 11.4;
      );
      =     L 0.0;
      A     L 0.0;
      FP    M 1000.3;
      S     Q 64.1;
      A     L 0.0;
      A     Q 64.1;
      A(;
      O     I 64.1;
      O     M 29.4;
      );
      R     Q 64.1;
NETWORK
TITLE = Enable Coral Vacuum
      A     M 11.4;
      A     M 72.0;
      =     Q 17.0;
NETWORK
TITLE = Test Gas Arc Pilota
//Test Arco Gas
      A     M 11.2;
      A     M 32.2;
      O;
      A     M 11.4;
      A     M 52.4;
      =     Q 17.7;
NETWORK
TITLE = Reset
//bit DI0 Select Scene TeleCam
      A     M 1.1;
      A(;
      O     M 90.1;
      O     M 90.3;
      );
      A     T 47;
      =     Q 64.3;
NETWORK
TITLE = DI1
//bit DI1 Select Scene TeleCam
      A     M 1.1;
      A(;
      O     M 90.2;
      O     M 90.3;
      );
      A     T 47;
      =     Q 64.4;
NETWORK
TITLE = DI1
//Select Scene Cam
      A     M 1.1;
      =     L 0.0;
      A     L 0.0;
      A     T 47;
      =     Q 65.2;
      A     L 0.0;
      A     T 47;
      =     Q 65.4;
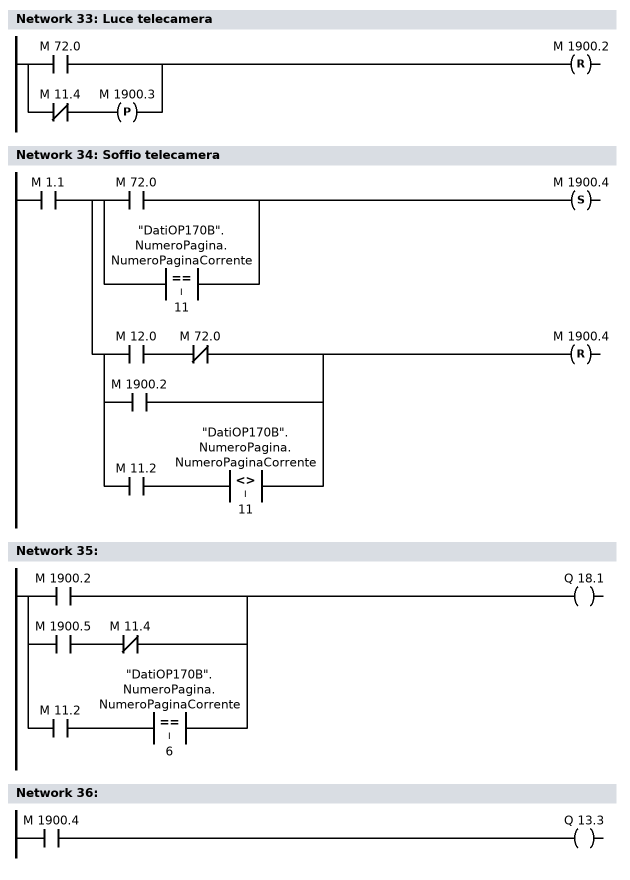
NETWORK
TITLE = Luce telecamera
      O     M 72.0;
      O(;
      AN    M 11.4;
      FP    M 1900.3;
      );
      R     M 1900.2;
NETWORK
TITLE = Soffio telecamera
      A     M 1.1;
      =     L 0.0;
      A     L 0.0;
      A(;
      O     M 72.0;
      O(;
      L     "DatiOP170B".NumeroPagina.NumeroPaginaCorrente;
      L     11;
      ==I;
      );
      );
      S     M 1900.4;
      A     L 0.0;
      A(;
      A     M 12.0;
      AN    M 72.0;
      O     M 1900.2;
      O;
      A     M 11.2;
      A(;
      L     "DatiOP170B".NumeroPagina.NumeroPaginaCorrente;
      L     11;
      <>I;
      );
      );
      R     M 1900.4;
NETWORK
TITLE =
      O     M 1900.2;
      O;
      A     M 1900.5;
      AN    M 11.4;
      O;
      A     M 11.2;
      A(;
      L     "DatiOP170B".NumeroPagina.NumeroPaginaCorrente;
      L     6;
      ==I;
      );
      =     Q 18.1;
NETWORK
TITLE =
      A     M 1900.4;
      =     Q 13.3;
END_FUNCTION

FUNCTION "FC19 - REPOSITIONING" : VOID	// FC 19
TITLE = Repositioning management
VERSION : 0.1
BEGIN
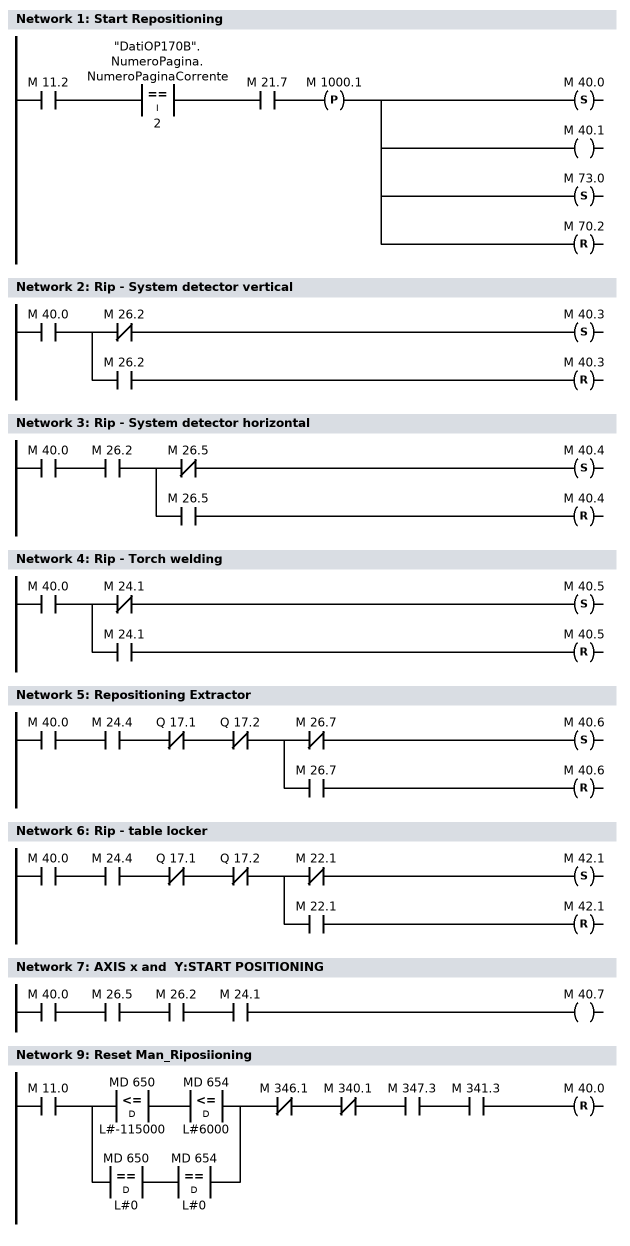
NETWORK
TITLE = Start Repositioning
      A     M 11.2;
      A(;
      L     "DatiOP170B".NumeroPagina.NumeroPaginaCorrente;
      L     2;
      ==I;
      );
      A     M 21.7;
      FP    M 1000.1;
      S     M 40.0;
      =     M 40.1;
      S     M 73.0;
      R     M 70.2;
NETWORK
TITLE = Rip - System detector vertical
//ripositioning Table
      A     M 40.0;
      =     L 0.0;
      A     L 0.0;
      AN    M 26.2;
      S     M 40.3;
      A     L 0.0;
      A     M 26.2;
      R     M 40.3;
NETWORK
TITLE = Rip - System detector horizontal
//ripositioning Table
      A     M 40.0;
      A     M 26.2;
      =     L 0.0;
      A     L 0.0;
      AN    M 26.5;
      S     M 40.4;
      A     L 0.0;
      A     M 26.5;
      R     M 40.4;
NETWORK
TITLE = Rip - Torch welding
//ripositioning Table
      A     M 40.0;
      =     L 0.0;
      A     L 0.0;
      AN    M 24.1;
      S     M 40.5;
      A     L 0.0;
      A     M 24.1;
      R     M 40.5;
NETWORK
TITLE = Repositioning Extractor
      A     M 40.0;
      A     M 24.4;
      AN    Q 17.1;
      AN    Q 17.2;
      =     L 0.0;
      A     L 0.0;
      AN    M 26.7;
      S     M 40.6;
      A     L 0.0;
      A     M 26.7;
      R     M 40.6;
NETWORK
TITLE = Rip - table locker
      A     M 40.0;
      A     M 24.4;
      AN    Q 17.1;
      AN    Q 17.2;
      =     L 0.0;
      A     L 0.0;
      AN    M 22.1;
      S     M 42.1;
      A     L 0.0;
      A     M 22.1;
      R     M 42.1;
NETWORK
TITLE = AXIS x and  Y:START POSITIONING
      A     M 40.0;
      A     M 26.5;
      A     M 26.2;
      A     M 24.1;
      =     M 40.7;
NETWORK
TITLE = Reset Man_Riposiioning
//      U     "START_POS"
//      U(    
//      U(    
//      L     "MD650"
//      L     L#-115000
//      <=D   
//      )     
//      U(    
//      L     "MD654"
//      L     L#6000
//      <=D   
//      )     
//      O     
//      U(    
//      L     "MD650"
//      L     L#0
//      ==I   
//      )     
//      U(    
//      L     "MD654"
//      L     L#0
//      ==I   
//      )     
//      )     
//      UN    "M346.1"
//      UN    "M340.1"
//      U     "M347.3"
//      U     "M341.3"
//      R     "M40.0"
NETWORK
TITLE = Reset Man_Riposiioning
      A     M 11.0;
      A(;
      A(;
      L     MD 650;
      L     L#-115000;
      <=D;
      );
      A(;
      L     MD 654;
      L     L#6000;
      <=D;
      );
      O;
      A(;
      L     MD 650;
      L     L#0;
      ==D;
      );
      A(;
      L     MD 654;
      L     L#0;
      ==D;
      );
      );
      AN    M 346.1;
      AN    M 340.1;
      A     M 347.3;
      A     M 341.3;
      R     M 40.0;
NETWORK
TITLE =
END_FUNCTION

FUNCTION "FC50 - TEACH-IN" : VOID	// FC 50
TITLE = TEACH_IN
VERSION : 0.1
BEGIN
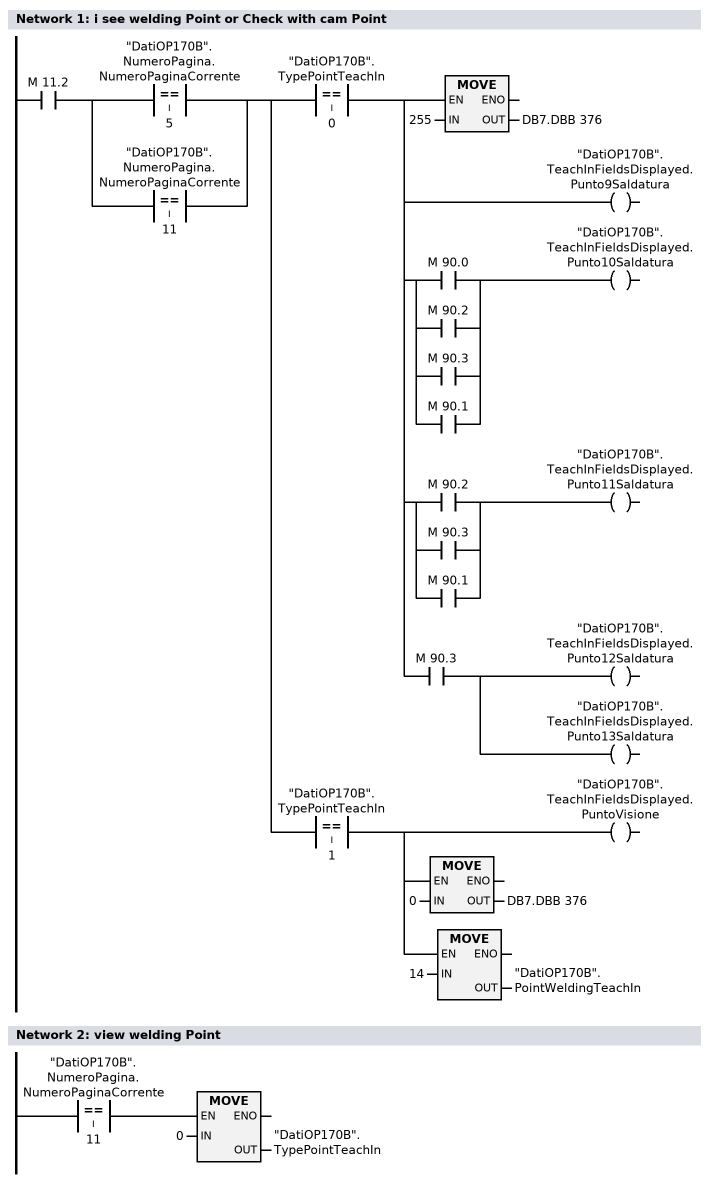
NETWORK
TITLE = i see welding Point or Check with cam Point
      A     M 11.2;
      A(;
      O(;
      L     "DatiOP170B".NumeroPagina.NumeroPaginaCorrente;
      L     5;
      ==I;
      );
      O(;
      L     "DatiOP170B".NumeroPagina.NumeroPaginaCorrente;
      L     11;
      ==I;
      );
      );
      =     L 0.0;
      A     L 0.0;
      A(;
      L     "DatiOP170B".TypePointTeachIn;
      L     0;
      ==I;
      );
      =     L 0.1;
      A     L 0.1;
      JNB   _001;
      L     255;
      T     DB7.DBB 376;
_001: NOP   0;
      A     L 0.1;
      BLD   102;
      =     "DatiOP170B".TeachInFieldsDisplayed.Punto9Saldatura;
      A     L 0.1;
      A(;
      O     M 90.0;
      O     M 90.2;
      O     M 90.3;
      O     M 90.1;
      );
      =     "DatiOP170B".TeachInFieldsDisplayed.Punto10Saldatura;
      A     L 0.1;
      A(;
      O     M 90.2;
      O     M 90.3;
      O     M 90.1;
      );
      =     "DatiOP170B".TeachInFieldsDisplayed.Punto11Saldatura;
      A     L 0.1;
      A     M 90.3;
      =     "DatiOP170B".TeachInFieldsDisplayed.Punto12Saldatura;
      =     "DatiOP170B".TeachInFieldsDisplayed.Punto13Saldatura;
      A     L 0.0;
      A(;
      L     "DatiOP170B".TypePointTeachIn;
      L     1;
      ==I;
      );
      =     L 0.1;
      A     L 0.1;
      BLD   102;
      =     "DatiOP170B".TeachInFieldsDisplayed.PuntoVisione;
      A     L 0.1;
      JNB   _002;
      L     0;
      T     DB7.DBB 376;
_002: NOP   0;
      A     L 0.1;
      JNB   _003;
      L     14;
      T     "DatiOP170B".PointWeldingTeachIn;
_003: NOP   0;
NETWORK
TITLE = view welding Point
      A(;
      L     "DatiOP170B".NumeroPagina.NumeroPaginaCorrente;
      L     11;
      ==I;
      );
      JNB   _004;
      L     0;
      T     "DatiOP170B".TypePointTeachIn;
_004: NOP   0;
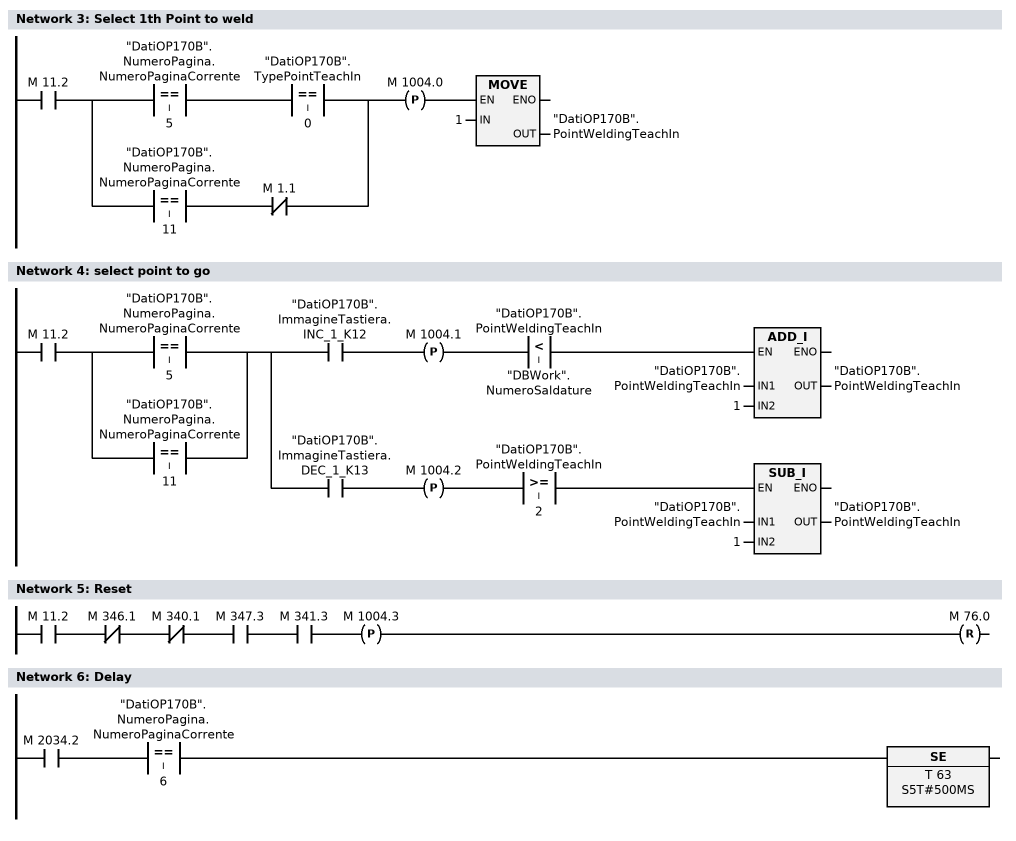
NETWORK
TITLE = Select 1th Point to weld
      A     M 11.2;
      A(;
      A(;
      L     "DatiOP170B".NumeroPagina.NumeroPaginaCorrente;
      L     5;
      ==I;
      );
      A(;
      L     "DatiOP170B".TypePointTeachIn;
      L     0;
      ==I;
      );
      O;
      A(;
      L     "DatiOP170B".NumeroPagina.NumeroPaginaCorrente;
      L     11;
      ==I;
      );
      AN    M 1.1;
      );
      FP    M 1004.0;
      JNB   _005;
      L     1;
      T     "DatiOP170B".PointWeldingTeachIn;
_005: NOP   0;
NETWORK
TITLE = select point to go
      A     M 11.2;
      A(;
      O(;
      L     "DatiOP170B".NumeroPagina.NumeroPaginaCorrente;
      L     5;
      ==I;
      );
      O(;
      L     "DatiOP170B".NumeroPagina.NumeroPaginaCorrente;
      L     11;
      ==I;
      );
      );
      =     L 0.0;
      A     L 0.0;
      A     "DatiOP170B".ImmagineTastiera.INC_1_K12;
      FP    M 1004.1;
      A(;
      L     "DatiOP170B".PointWeldingTeachIn;
      L     "DBWork".NumeroSaldature;
      <I;
      );
      JNB   _006;
      L     "DatiOP170B".PointWeldingTeachIn;
      L     1;
      +I;
      T     "DatiOP170B".PointWeldingTeachIn;
_006: NOP   0;
      A     L 0.0;
      A     "DatiOP170B".ImmagineTastiera.DEC_1_K13;
      FP    M 1004.2;
      A(;
      L     "DatiOP170B".PointWeldingTeachIn;
      L     2;
      >=I;
      );
      JNB   _007;
      L     "DatiOP170B".PointWeldingTeachIn;
      L     1;
      -I;
      T     "DatiOP170B".PointWeldingTeachIn;
_007: NOP   0;
NETWORK
TITLE = Reset
      A     M 11.2;
      AN    M 346.1;
      AN    M 340.1;
      A     M 347.3;
      A     M 341.3;
      FP    M 1004.3;
      R     M 76.0;
NETWORK
TITLE = Delay
      A     M 2034.2;
      A(;
      L     "DatiOP170B".NumeroPagina.NumeroPaginaCorrente;
      L     6;
      ==I;
      );
      L     S5T#500MS;
      SE    T 63;
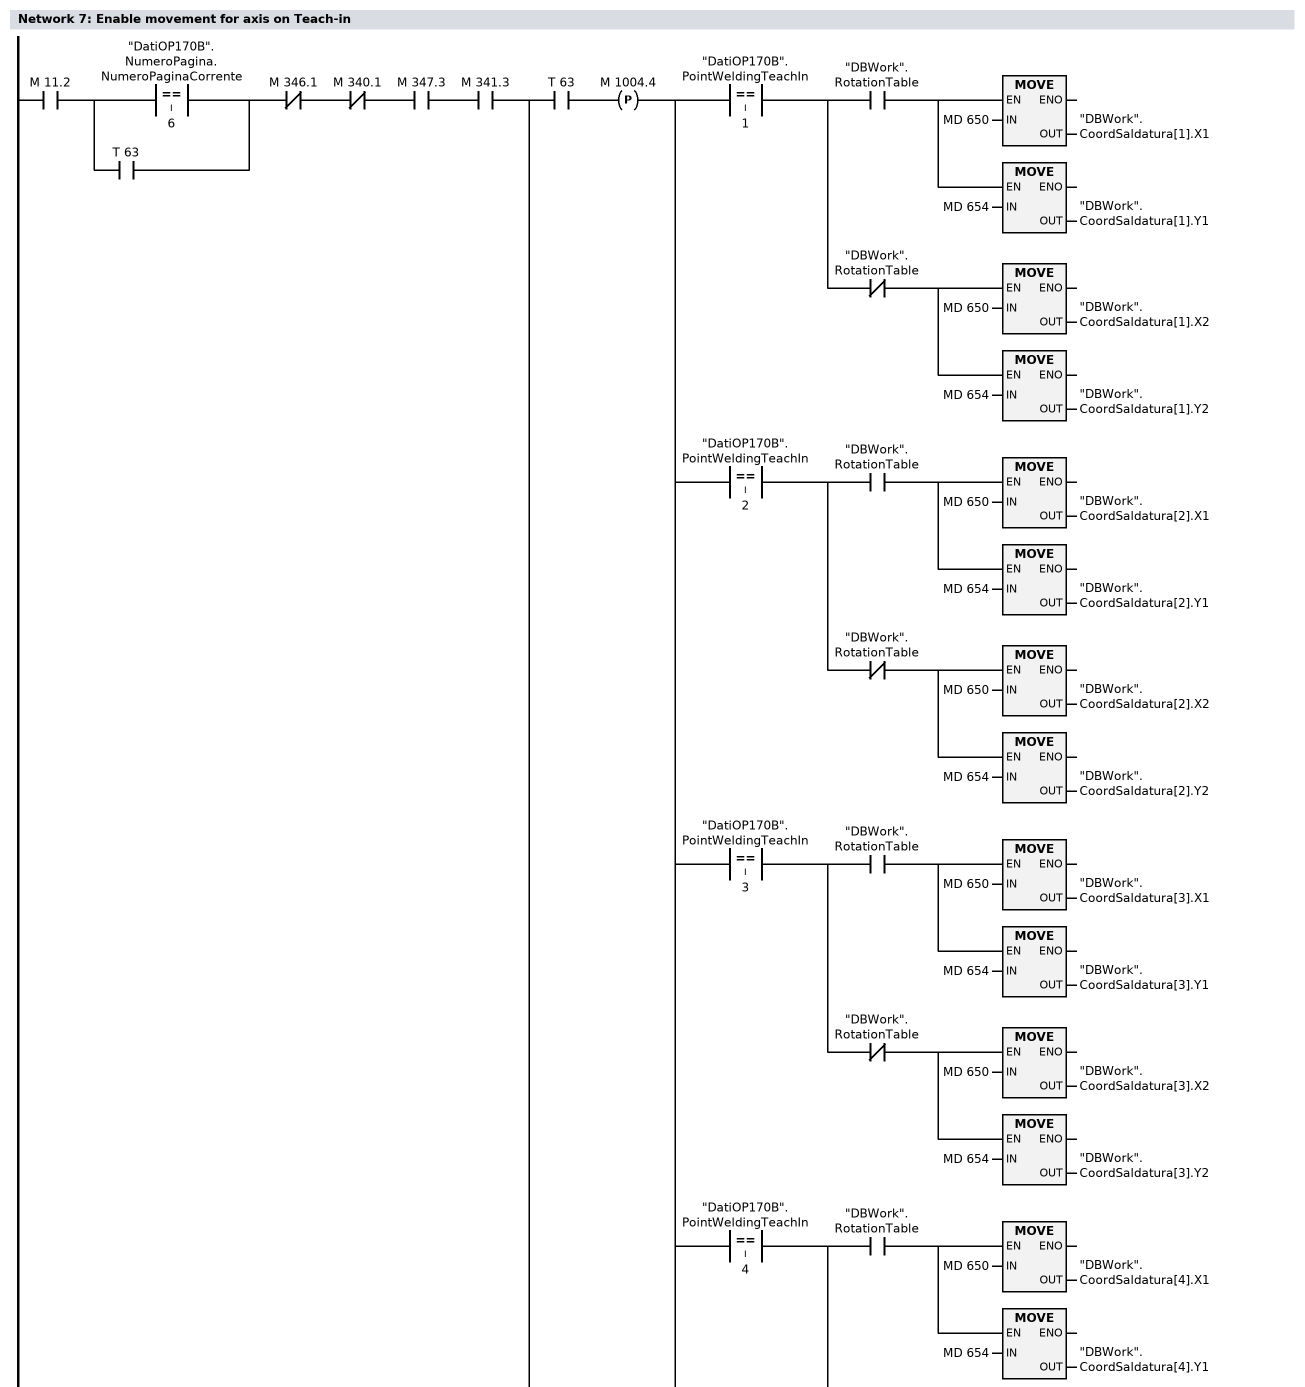
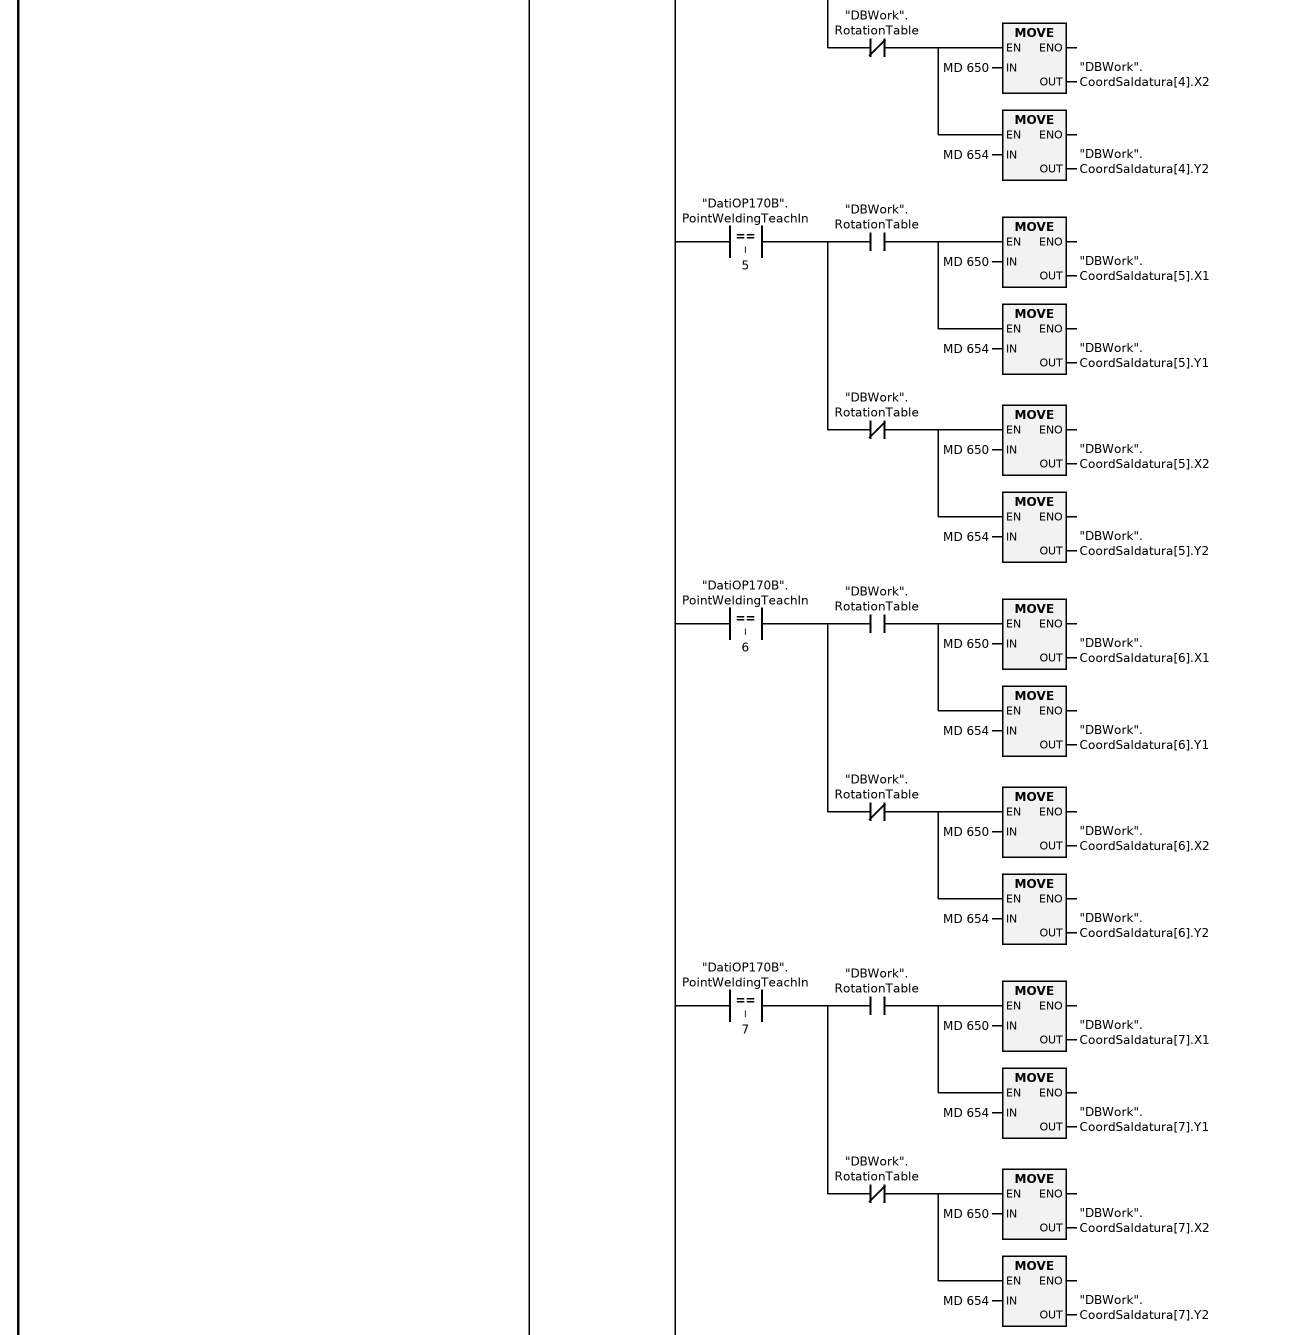
